// TIA Portal project "new" (V15.1)

(* hardware
DEVICE "S71500/ET200MP station_1"  S7-1500 station
   slot 0: "导轨_0"  Rack  6ES7 590-1***0-0AA0
   slot 1: "jvzihengtian"  CPU 1512C-1 PN  6ES7 512-1CK01-0AB0  V2.5
      slot 3: "CPU 显示_1"  6ES7591-1AA00-0AA0
DEVICE "DESKTOP-H96SFRB"  SIMATIC PC station
   slot 0: "SIMATIC PC station"  Rail  SIMATIC PC-Station  V1.0
      slot 125: "Stationmanager"  Station_Manager  V6.0.4
   slot 1: "IE general_1"  IE General  IE_CP  V8.2.0
   slot 2: "HMI_RT_1"  WinCC RT Advanced  6AV2 104-0xxxx-xxxx  15.1.0.0
      slot 33792: "主机接口"  Host interface
*)

// ===== PLC "jvzihengtian"  CPU 1512C-1 PN =====

DATA_BLOCK "输入变量"   // DB1
{ S7_Optimized_Access := 'FALSE' }
VERSION : 0.1
   VAR
      "1层上行呼梯按钮" : Bool;
      "2层上行呼梯按钮" : Bool;
      "3层上行呼梯按钮" : Bool;
      "4层上行呼梯按钮" : Bool;
      "5层上行呼梯按钮" : Bool;
      "2层下行呼梯按钮" : Bool;
      "3层下行呼梯按钮" : Bool;
      "4层下行呼梯按钮" : Bool;
      "5层下行呼梯按钮" : Bool;
      "6层下行呼梯按钮" : Bool;
      "1号梯轿内选层按钮1" : Bool;
      "1号梯轿内选层按钮2" : Bool;
      "1号梯轿内选层按钮3" : Bool;
      "1号梯轿内选层按钮4" : Bool;
      "1号梯轿内选层按钮5" : Bool;
      "1号梯轿内选层按钮6" : Bool;
      "1号梯轿内开门按钮" : Bool;
      "1号梯轿内关门按钮" : Bool;
      "1号梯光幕信号" : Bool;
      "1号梯检修信号" : Bool;
      "1号梯轿厢门锁信号" : Bool;
      "1号梯1楼层门锁信号" : Bool;
      "1号梯2楼层门锁信号" : Bool;
      "1号梯3楼层门锁信号" : Bool;
      "1号梯4楼层门锁信号" : Bool;
      "1号梯5楼层门锁信号" : Bool;
      "1号梯6楼层门锁信号" : Bool;
      "1号梯开门到位" : Bool;
      "1号梯关门到位" : Bool;
      "1号梯上平层信号" : Bool;
      "1号梯下平层信号" : Bool;
      "1号梯上端站第1限位" : Bool;
      "1号梯上端站第2限位" : Bool;
      "1号梯下端站第1限位" : Bool;
      "1号梯下端站第2限位" : Bool;
      自动运行信号 : Bool;
      "1号梯当前载重量" : Word;
   END_VAR
BEGIN
END_DATA_BLOCK

DATA_BLOCK "输出变量"   // DB2
{ S7_Optimized_Access := 'FALSE' }
VERSION : 0.1
   VAR
      "1层上行呼梯按钮指示灯" : Bool;
      "2层上行呼梯按钮指示灯" : Bool;
      "3层上行呼梯按钮指示灯" : Bool;
      "4层上行呼梯按钮指示灯" : Bool;
      "5层上行呼梯按钮指示灯" : Bool;
      "2层下行呼梯按钮指示灯" : Bool;
      "3层下行呼梯按钮指示灯" : Bool;
      "4层下行呼梯按钮指示灯" : Bool;
      "5层下行呼梯按钮指示灯" : Bool;
      "6层下行呼梯按钮指示灯" : Bool;
      "1号梯1层按钮指示灯" : Bool;
      "1号梯2层按钮指示灯" : Bool;
      "1号梯3层按钮指示灯" : Bool;
      "1号梯4层按钮指示灯" : Bool;
      "1号梯5层按钮指示灯" : Bool;
      "1号梯6层按钮指示灯" : Bool;
      "1号梯LEDa" : Bool;
      "1号梯LEDb" : Bool;
      "1号梯LEDc" : Bool;
      "1号梯LEDd" : Bool;
      "1号梯LEDe" : Bool;
      "1号梯LEDf" : Bool;
      "1号梯LEDg" : Bool;
      "1号梯上行指示" : Bool;
      "1号梯下行指示" : Bool;
      "1号梯故障指示" : Bool;
      "1号梯照明指示" : Bool;
      "1号梯风扇指示" : Bool;
      "1号梯满载指示" : Bool;
      "1号梯电机启动信号" : Bool := false;
      "1号梯上行接触器" : Bool;
      "1号梯下行接触器" : Bool;
      "1号梯高速接触器" : Bool;
      "1号梯低速接触器" : Bool;
      "1号梯开门继电器" : Bool;
      "1号梯关门继电器" : Bool;
      "1号梯1级减速制动" : Bool;
      "1号梯2级减速制动" : Bool;
      "1号梯3级减速制动" : Bool;
      准备就绪信号 : Bool := false;
   END_VAR
BEGIN
END_DATA_BLOCK

DATA_BLOCK "一梯辅助变量"   // DB29
{ S7_Optimized_Access := 'FALSE' }
VERSION : 0.1
   VAR
      "1层上呼tag" : Bool;
      "1层上呼开门tag" : Bool;
      "1梯关门标志" : Bool;
      "2层上呼tag" : Bool;
      "2层上呼开门tag" : Bool;
      "2层下呼tag" : Bool;
      "2层下呼开门tag" : Bool;
      "3层上呼tag" : Bool;
      "3层上呼开门tag" : Bool;
      "3层下呼tag" : Bool;
      "3层下呼开门tag" : Bool;
      "4层上呼tag" : Bool;
      "4层上呼开门tag" : Bool;
      "4层下呼tag" : Bool;
      "4层下呼开门tag" : Bool;
      "5层上呼tag" : Bool;
      "5层上呼开门tag" : Bool;
      "5层下呼tag" : Bool;
      "5层下呼开门tag" : Bool;
      "6层下呼tag" : Bool;
      "6层下呼开门tag" : Bool;
      T总延时 : Bool;
      一号梯内选1 : Bool;
      一号梯内选2 : Bool;
      一号梯内选3 : Bool;
      一号梯内选4 : Bool;
      一号梯内选5 : Bool;
      一号梯内选6 : Bool;
      一号梯初始化 : Bool;
      一号梯楼层数 : Int := 1;
      一号梯自动运行脉冲检测 : Bool;
      一层上呼标志 : Bool;
      三层上呼标志 : Bool;
      三层下呼标志 : Bool;
      "上行1，下行0，默认下" : Bool := false;
      上行标志 : Bool;
      下行标志 : Bool;
      二层上呼标志 : Bool;
      二层下呼标志 : Bool;
      五层上呼标志 : Bool;
      五层下呼标志 : Bool;
      停在1层 : Bool;
      停在2层 : Bool;
      停在3层 : Bool;
      停在4层 : Bool;
      停在5层 : Bool;
      停在6层 : Bool;
      停层信号 : Bool;
      停层关门辅助 : Bool;
      停层开门 : Bool;
      停层时上下呼开门 : Bool;
      光幕信号标志 : Bool;
      六层下呼标志 : Bool;
      关门异常重新开门 : Bool;
      关门按钮标志 : Bool;
      内选1tag : Bool;
      内选2tag : Bool;
      内选3tag : Bool;
      内选4tag : Bool;
      内选5tag : Bool;
      内选6tag : Bool;
      内选停层信号 : Bool;
      初始化上行控制 : Bool;
      初始化下行控制 : Bool;
      初始化变量1 : Bool;
      初始化变量2 : Bool;
      初始化已停层 : Bool;
      初始化平层tag : Bool;
      初始化楼层数检测 : Bool;
      到1限 : Bool;
      四层上呼标志 : Bool;
      四层下呼标志 : Bool;
      外呼停层信号 : Bool;
      延时关门辅助 : Bool;
      延时自动关门 : Bool;
      开门完成标志 : Bool;
      开门异常重新关门 : Bool;
      开门按钮标志 : Bool;
      开门标志 : Bool;
      有人出不关门 : Bool;
      楼层计数平层tag1 : Bool;
      楼层计数平层tag2 : Bool;
      超载异常强制关门 : Bool;
      超重信号 : Bool;
      超重信号tag : Bool;
      超重信号标志 : Bool;
      超重次数 : Int;
      超重次数初值 : Int;
      超重次数变化值 : Int;
      信号状态连接1 : Bool;
      载重量初值 : Word := 16#0000;
      载重变化次数计数 : Int := 0;
      载重变化一次 : Bool;
      载重变化一次tag : Bool;
      "1梯初始化到几层" : Int;
      上行1 : Bool;
      下行1 : Bool;
      上行1关 : Bool;
      下行1关 : Bool;
      上行状态检查 : Bool;
      下行状态检查 : Bool;
      上行接触器tag : Bool;
      下行接触器tag : Bool;
      上行接触器1到0 : Bool;
      下行接触器1到0 : Bool;
      开门按钮tag : Bool;
      关门按钮tag : Bool;
      光幕tag : Bool;
      "1层保护1" : Bool;
      "1层保护2" : Bool;
      "6层保护1" : Bool;
      "6层保护2" : Bool;
      内选1预消除 : Bool;
      载重量最大允许值 : Int := 13129;
      门锁状态 : Bool;
      载重变化次数max : Int := 16;
      外呼响应载重量限值 : Int := 12438;
   END_VAR
BEGIN
END_DATA_BLOCK

// folder: System blocks/Program resources

DATA_BLOCK "三级减速制动T总"   // DB3
{ S7_Optimized_Access := 'TRUE' }
AUTHOR : Simatic
FAMILY : IEC
NAME : IEC_TMR
VERSION : 1.0
// stored: InstanceOfName IEC_TIMER
"IEC_TIMER"
BEGIN
END_DATA_BLOCK

DATA_BLOCK "一级减速制动T1"   // DB4
{ S7_Optimized_Access := 'TRUE' }
AUTHOR : Simatic
FAMILY : IEC
NAME : IEC_TMR
VERSION : 1.0
// stored: InstanceOfName IEC_TIMER
"IEC_TIMER"
BEGIN
END_DATA_BLOCK

DATA_BLOCK "二级减速制动T2"   // DB5
{ S7_Optimized_Access := 'TRUE' }
AUTHOR : Simatic
FAMILY : IEC
NAME : IEC_TMR
VERSION : 1.0
// stored: InstanceOfName IEC_TIMER
"IEC_TIMER"
BEGIN
END_DATA_BLOCK

DATA_BLOCK "上下行复位脉冲"   // DB6
{ S7_Optimized_Access := 'TRUE' }
AUTHOR : Simatic
FAMILY : IEC
NAME : IEC_TMR
VERSION : 1.0
// stored: InstanceOfName IEC_TIMER
"IEC_TIMER"
BEGIN
END_DATA_BLOCK

DATA_BLOCK "初始化平层延时"   // DB7
{ S7_Optimized_Access := 'TRUE' }
AUTHOR : Simatic
FAMILY : IEC
NAME : IEC_TMR
VERSION : 1.0
// stored: InstanceOfName IEC_TIMER
"IEC_TIMER"
BEGIN
END_DATA_BLOCK

DATA_BLOCK "三级减速制动T3"   // DB8
{ S7_Optimized_Access := 'TRUE' }
AUTHOR : Simatic
FAMILY : IEC
NAME : IEC_TMR
VERSION : 1.0
// stored: InstanceOfName IEC_TIMER
"IEC_TIMER"
BEGIN
END_DATA_BLOCK

DATA_BLOCK "关断延时1"   // DB9
{ S7_Optimized_Access := 'TRUE' }
AUTHOR : Simatic
FAMILY : IEC
NAME : IEC_TMR
VERSION : 1.0
// stored: InstanceOfName IEC_TIMER
"IEC_TIMER"
BEGIN
END_DATA_BLOCK

DATA_BLOCK "停层完成延时辅助"   // DB11
{ S7_Optimized_Access := 'TRUE' }
AUTHOR : Simatic
FAMILY : IEC
NAME : IEC_TMR
VERSION : 1.0
// stored: InstanceOfName IEC_TIMER
"IEC_TIMER"
BEGIN
END_DATA_BLOCK

DATA_BLOCK "门锁好复位延时"   // DB12
{ S7_Optimized_Access := 'TRUE' }
AUTHOR : Simatic
FAMILY : IEC
NAME : IEC_TMR
VERSION : 1.0
// stored: InstanceOfName IEC_TIMER
"IEC_TIMER"
BEGIN
END_DATA_BLOCK

DATA_BLOCK "开到位延时"   // DB13
{ S7_Optimized_Access := 'TRUE' }
AUTHOR : Simatic
FAMILY : IEC
NAME : IEC_TMR
VERSION : 1.0
// stored: InstanceOfName IEC_TIMER
"IEC_TIMER"
BEGIN
END_DATA_BLOCK

DATA_BLOCK "关断延时2"   // DB14
{ S7_Optimized_Access := 'TRUE' }
AUTHOR : Simatic
FAMILY : IEC
NAME : IEC_TMR
VERSION : 1.0
// stored: InstanceOfName IEC_TIMER
"IEC_TIMER"
BEGIN
END_DATA_BLOCK

DATA_BLOCK "关断延时3"   // DB15
{ S7_Optimized_Access := 'TRUE' }
AUTHOR : Simatic
FAMILY : IEC
NAME : IEC_TMR
VERSION : 1.0
// stored: InstanceOfName IEC_TIMER
"IEC_TIMER"
BEGIN
END_DATA_BLOCK

DATA_BLOCK "关断延时4"   // DB16
{ S7_Optimized_Access := 'TRUE' }
AUTHOR : Simatic
FAMILY : IEC
NAME : IEC_TMR
VERSION : 1.0
// stored: InstanceOfName IEC_TIMER
"IEC_TIMER"
BEGIN
END_DATA_BLOCK

DATA_BLOCK "关断延时5"   // DB17
{ S7_Optimized_Access := 'TRUE' }
AUTHOR : Simatic
FAMILY : IEC
NAME : IEC_TMR
VERSION : 1.0
// stored: InstanceOfName IEC_TIMER
"IEC_TIMER"
BEGIN
END_DATA_BLOCK

DATA_BLOCK "关断延时6"   // DB18
{ S7_Optimized_Access := 'TRUE' }
AUTHOR : Simatic
FAMILY : IEC
NAME : IEC_TMR
VERSION : 1.0
// stored: InstanceOfName IEC_TIMER
"IEC_TIMER"
BEGIN
END_DATA_BLOCK

DATA_BLOCK "关断延时7"   // DB19
{ S7_Optimized_Access := 'TRUE' }
AUTHOR : Simatic
FAMILY : IEC
NAME : IEC_TMR
VERSION : 1.0
// stored: InstanceOfName IEC_TIMER
"IEC_TIMER"
BEGIN
END_DATA_BLOCK

DATA_BLOCK "待载休眠计时"   // DB20
{ S7_Optimized_Access := 'TRUE' }
AUTHOR : Simatic
FAMILY : IEC
NAME : IEC_TMR
VERSION : 1.0
// stored: InstanceOfName IEC_TIMER
"IEC_TIMER"
BEGIN
END_DATA_BLOCK

DATA_BLOCK "关门时间"   // DB21
{ S7_Optimized_Access := 'TRUE' }
AUTHOR : Simatic
FAMILY : IEC
NAME : IEC_TMR
VERSION : 1.0
// stored: InstanceOfName IEC_TIMER
"IEC_TIMER"
BEGIN
END_DATA_BLOCK

DATA_BLOCK "关断延时8"   // DB22
{ S7_Optimized_Access := 'TRUE' }
AUTHOR : Simatic
FAMILY : IEC
NAME : IEC_TMR
VERSION : 1.0
// stored: InstanceOfName IEC_TIMER
"IEC_TIMER"
BEGIN
END_DATA_BLOCK

DATA_BLOCK "超重延时判断"   // DB23
{ S7_Optimized_Access := 'TRUE' }
AUTHOR : Simatic
FAMILY : IEC
NAME : IEC_TMR
VERSION : 1.0
// stored: InstanceOfName IEC_TIMER
"IEC_TIMER"
BEGIN
END_DATA_BLOCK

DATA_BLOCK "超载异常脉冲"   // DB24
{ S7_Optimized_Access := 'TRUE' }
AUTHOR : Simatic
FAMILY : IEC
NAME : IEC_TMR
VERSION : 1.0
// stored: InstanceOfName IEC_TIMER
"IEC_TIMER"
BEGIN
END_DATA_BLOCK

DATA_BLOCK "关断延时9"   // DB25
{ S7_Optimized_Access := 'TRUE' }
AUTHOR : Simatic
FAMILY : IEC
NAME : IEC_TMR
VERSION : 1.0
// stored: InstanceOfName IEC_TIMER
"IEC_TIMER"
BEGIN
END_DATA_BLOCK

DATA_BLOCK "低速启动延时"   // DB26
{ S7_Optimized_Access := 'TRUE' }
AUTHOR : Simatic
FAMILY : IEC
NAME : IEC_TMR
VERSION : 1.0
// stored: InstanceOfName IEC_TIMER
"IEC_TIMER"
BEGIN
END_DATA_BLOCK

DATA_BLOCK "关断延时10"   // DB27
{ S7_Optimized_Access := 'TRUE' }
AUTHOR : Simatic
FAMILY : IEC
NAME : IEC_TMR
VERSION : 1.0
// stored: InstanceOfName IEC_TIMER
"IEC_TIMER"
BEGIN
END_DATA_BLOCK

DATA_BLOCK "开门时间"   // DB28
{ S7_Optimized_Access := 'TRUE' }
AUTHOR : Simatic
FAMILY : IEC
NAME : IEC_TMR
VERSION : 1.0
// stored: InstanceOfName IEC_TIMER
"IEC_TIMER"
BEGIN
END_DATA_BLOCK

DATA_BLOCK "载重量比较"   // DB30
{ S7_Optimized_Access := 'TRUE' }
AUTHOR : Simatic
FAMILY : IEC
NAME : IEC_TMR
VERSION : 1.0
// stored: InstanceOfName IEC_TIMER
"IEC_TIMER"
BEGIN
END_DATA_BLOCK

DATA_BLOCK "采样、比较时间间隔"   // DB31
{ S7_Optimized_Access := 'TRUE' }
AUTHOR : Simatic
FAMILY : IEC
NAME : IEC_TMR
VERSION : 1.0
// stored: InstanceOfName IEC_TIMER
"IEC_TIMER"
BEGIN
END_DATA_BLOCK

DATA_BLOCK "载重量采样"   // DB32
{ S7_Optimized_Access := 'TRUE' }
AUTHOR : Simatic
FAMILY : IEC
NAME : IEC_TMR
VERSION : 1.0
// stored: InstanceOfName IEC_TIMER
"IEC_TIMER"
BEGIN
END_DATA_BLOCK

DATA_BLOCK "关断延时11"   // DB33
{ S7_Optimized_Access := 'TRUE' }
AUTHOR : Simatic
FAMILY : IEC
NAME : IEC_TMR
VERSION : 1.0
// stored: InstanceOfName IEC_TIMER
"IEC_TIMER"
BEGIN
END_DATA_BLOCK

DATA_BLOCK "IEC_Timer_0_DB_4"   // DB34
{ S7_Optimized_Access := 'TRUE' }
AUTHOR : Simatic
FAMILY : IEC
NAME : IEC_TMR
VERSION : 1.0
// stored: InstanceOfName IEC_TIMER
"IEC_TIMER"
BEGIN
END_DATA_BLOCK

DATA_BLOCK "关断延时12"   // DB35
{ S7_Optimized_Access := 'TRUE' }
AUTHOR : Simatic
FAMILY : IEC
NAME : IEC_TMR
VERSION : 1.0
// stored: InstanceOfName IEC_TIMER
"IEC_TIMER"
BEGIN
END_DATA_BLOCK

DATA_BLOCK "关断延时13"   // DB36
{ S7_Optimized_Access := 'TRUE' }
AUTHOR : Simatic
FAMILY : IEC
NAME : IEC_TMR
VERSION : 1.0
// stored: InstanceOfName IEC_TIMER
"IEC_TIMER"
BEGIN
END_DATA_BLOCK

DATA_BLOCK "关断延时14"   // DB37
{ S7_Optimized_Access := 'TRUE' }
AUTHOR : Simatic
FAMILY : IEC
NAME : IEC_TMR
VERSION : 1.0
// stored: InstanceOfName IEC_TIMER
"IEC_TIMER"
BEGIN
END_DATA_BLOCK

DATA_BLOCK "关断延时15"   // DB38
{ S7_Optimized_Access := 'TRUE' }
AUTHOR : Simatic
FAMILY : IEC
NAME : IEC_TMR
VERSION : 1.0
// stored: InstanceOfName IEC_TIMER
"IEC_TIMER"
BEGIN
END_DATA_BLOCK

DATA_BLOCK "关断延时16"   // DB39
{ S7_Optimized_Access := 'TRUE' }
AUTHOR : Simatic
FAMILY : IEC
NAME : IEC_TMR
VERSION : 1.0
// stored: InstanceOfName IEC_TIMER
"IEC_TIMER"
BEGIN
END_DATA_BLOCK

DATA_BLOCK "计数"   // DB40
{ S7_Optimized_Access := 'TRUE' }
AUTHOR : Simatic
FAMILY : IEC
NAME : CNTR
VERSION : 1.0
// stored: InstanceOfName IEC_COUNTER
"IEC_COUNTER"
BEGIN
END_DATA_BLOCK

DATA_BLOCK "内选错误消除限时"   // DB50
{ S7_Optimized_Access := 'TRUE' }
AUTHOR : Simatic
FAMILY : IEC
NAME : IEC_TMR
VERSION : 1.0
// stored: InstanceOfName IEC_TIMER
"IEC_TIMER"
BEGIN
END_DATA_BLOCK

DATA_BLOCK "消除标志复位"   // DB51
{ S7_Optimized_Access := 'TRUE' }
AUTHOR : Simatic
FAMILY : IEC
NAME : IEC_TMR
VERSION : 1.0
// stored: InstanceOfName IEC_TIMER
"IEC_TIMER"
BEGIN
END_DATA_BLOCK

DATA_BLOCK "消除延时"   // DB52
{ S7_Optimized_Access := 'TRUE' }
AUTHOR : Simatic
FAMILY : IEC
NAME : IEC_TMR
VERSION : 1.0
// stored: InstanceOfName IEC_TIMER
"IEC_TIMER"
BEGIN
END_DATA_BLOCK

// folder: (top level)

FUNCTION "初始化下行" : Void   // FC1, LAD
{ S7_Optimized_Access := 'TRUE' }
VERSION : 0.1
   VAR_TEMP   // added for the SCL form of the ladder/FBD networks
      _w1 : Bool;
   END_VAR
BEGIN

REGION Network 1: 下行初始化
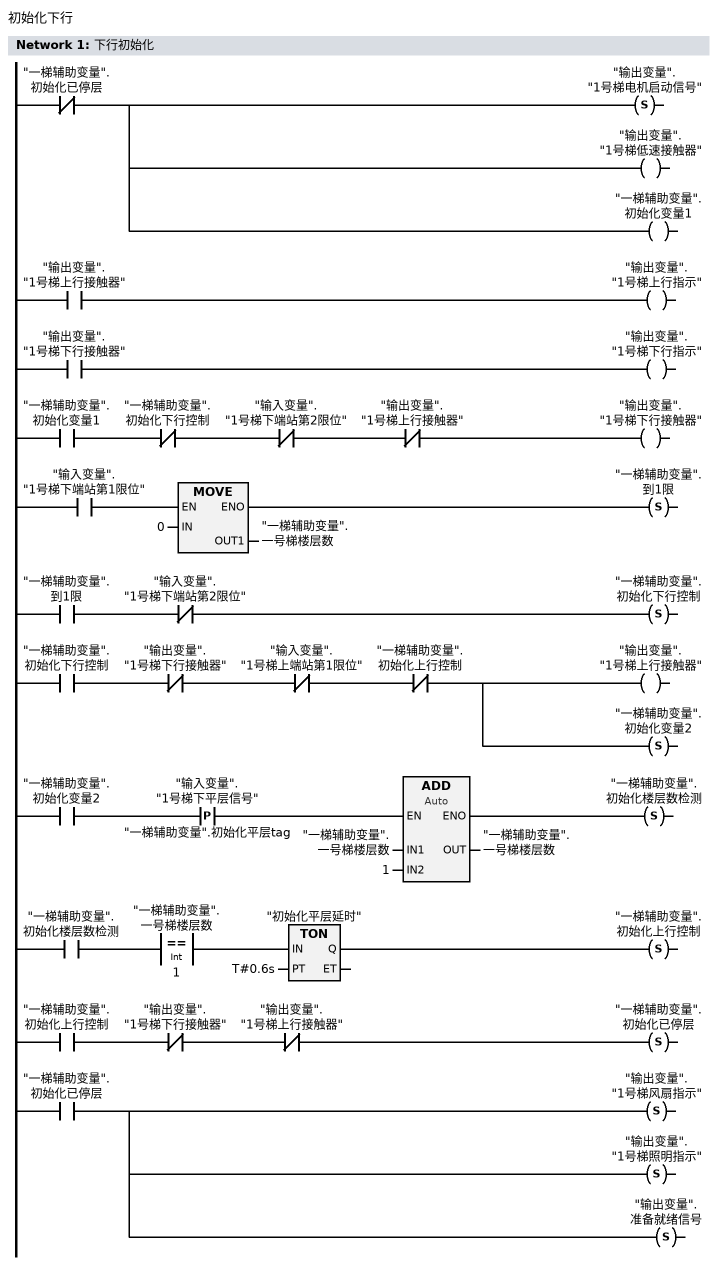
   IF NOT "一梯辅助变量".初始化已停层 THEN "输出变量"."1号梯电机启动信号" := TRUE; END_IF;
   "输出变量"."1号梯低速接触器" := NOT "一梯辅助变量".初始化已停层;
   "一梯辅助变量".初始化变量1 := NOT "一梯辅助变量".初始化已停层;
   "输出变量"."1号梯上行指示" := "输出变量"."1号梯上行接触器";
   "输出变量"."1号梯下行指示" := "输出变量"."1号梯下行接触器";
   "输出变量"."1号梯下行接触器" := "一梯辅助变量".初始化变量1 AND NOT "一梯辅助变量".初始化下行控制 AND NOT "输入变量"."1号梯下端站第2限位" AND NOT "输出变量"."1号梯上行接触器";
   IF "输入变量"."1号梯下端站第1限位" THEN
       "一梯辅助变量".一号梯楼层数 := 0;
       "一梯辅助变量".到1限 := TRUE;
   END_IF;
   IF "一梯辅助变量".到1限 AND NOT "输入变量"."1号梯下端站第2限位" THEN "一梯辅助变量".初始化下行控制 := TRUE; END_IF;
   "输出变量"."1号梯上行接触器" := "一梯辅助变量".初始化下行控制 AND NOT "输出变量"."1号梯下行接触器" AND NOT "输入变量"."1号梯上端站第1限位" AND NOT "一梯辅助变量".初始化上行控制;
   IF "输出变量"."1号梯上行接触器" THEN "一梯辅助变量".初始化变量2 := TRUE; END_IF;
   #_w1 := "一梯辅助变量".初始化变量2 AND "输入变量"."1号梯下平层信号" AND NOT "一梯辅助变量".初始化平层tag;   // rising edge of "输入变量"."1号梯下平层信号"
   "一梯辅助变量".初始化平层tag := "输入变量"."1号梯下平层信号";
   IF #_w1 THEN
       "一梯辅助变量".一号梯楼层数 := "一梯辅助变量".一号梯楼层数 + 1;
       "一梯辅助变量".初始化楼层数检测 := TRUE;
   END_IF;
   "初始化平层延时".TON(IN := "一梯辅助变量".初始化楼层数检测 AND ("一梯辅助变量".一号梯楼层数 = 1), PT := T#0.6s);
   IF "初始化平层延时".Q THEN "一梯辅助变量".初始化上行控制 := TRUE; END_IF;
   IF "一梯辅助变量".初始化上行控制 AND NOT "输出变量"."1号梯下行接触器" AND NOT "输出变量"."1号梯上行接触器" THEN
       "一梯辅助变量".初始化已停层 := TRUE;
   END_IF;
   IF "一梯辅助变量".初始化已停层 THEN
       "输出变量"."1号梯风扇指示" := TRUE;
       "输出变量"."1号梯照明指示" := TRUE;
       "输出变量".准备就绪信号 := TRUE;
   END_IF;
END_REGION
END_FUNCTION

FUNCTION "呼梯信号" : Void   // FC2, LAD
{ S7_Optimized_Access := 'TRUE' }
VERSION : 0.1
   VAR_TEMP   // added for the SCL form of the ladder/FBD networks
      _w1 : Bool;
      _w2 : Bool;
      _w3 : Bool;
      _w4 : Bool;
      _w5 : Bool;
      _w6 : Bool;
      _w7 : Bool;
      _w8 : Bool;
      _w9 : Bool;
      _w10 : Bool;
      _w11 : Bool;
      _w12 : Bool;
   END_VAR
BEGIN

REGION Network 1: 外呼灯
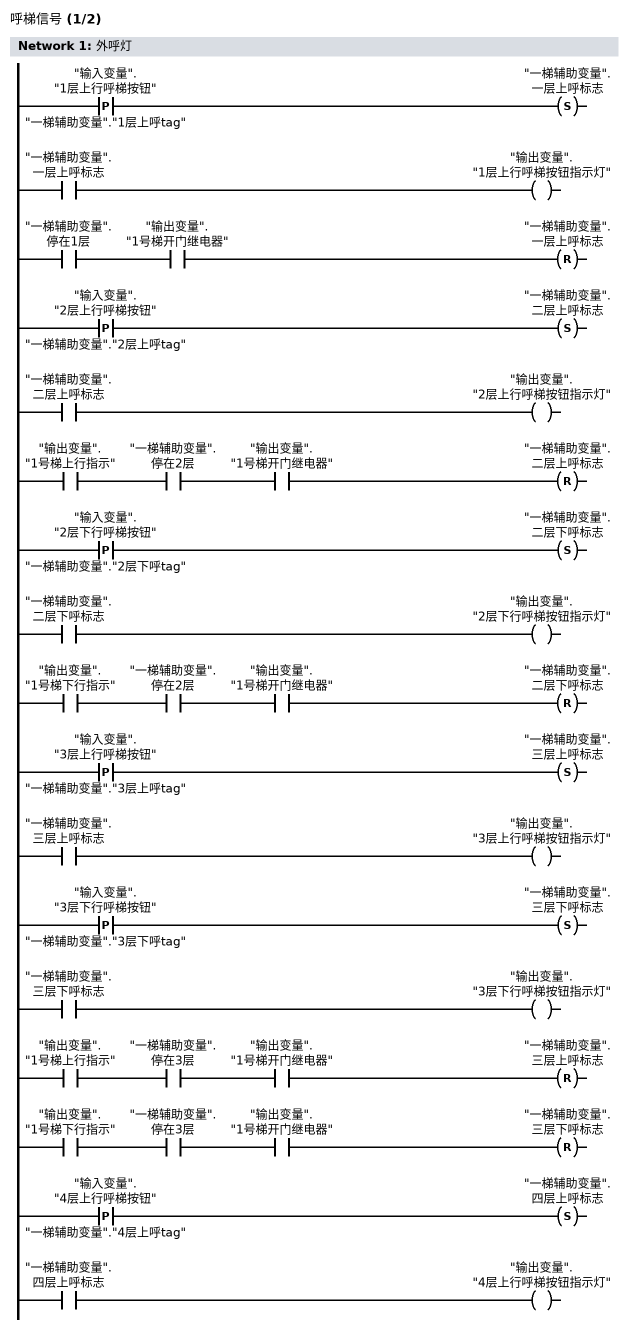
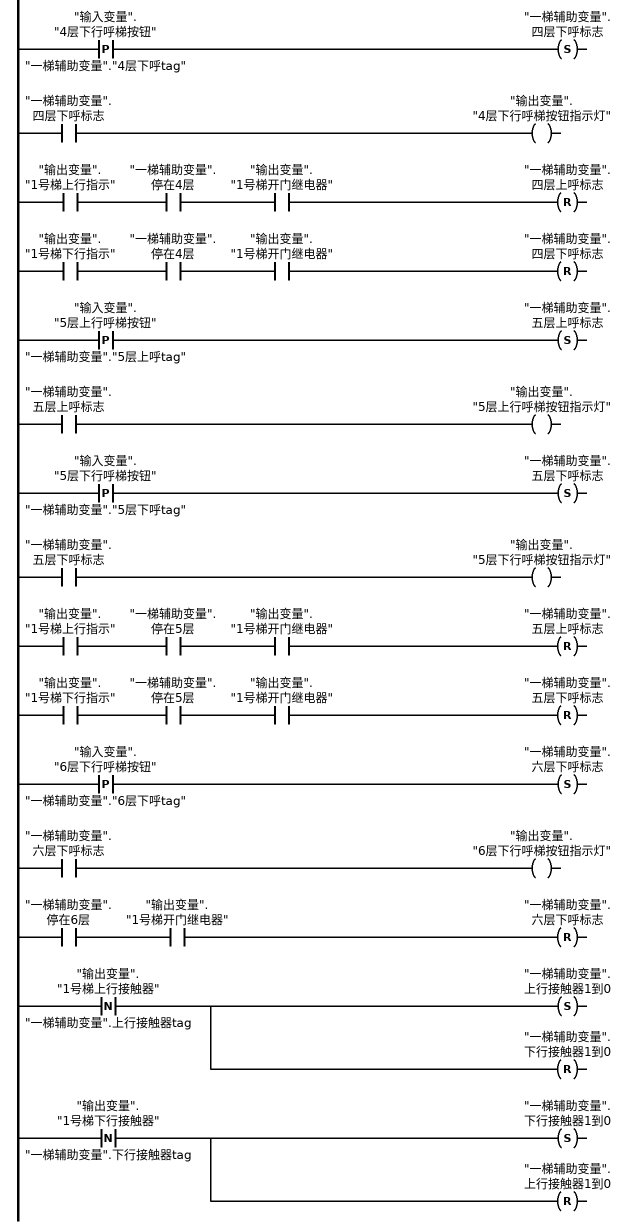
   RUNG wire#powerrail
      P_Contact(operand := "输入变量"."1层上行呼梯按钮", bit := "一梯辅助变量"."1层上呼tag")
      S_Coil( "一梯辅助变量".一层上呼标志 )
   END_RUNG
   RUNG wire#powerrail
      Contact( "一梯辅助变量".一层上呼标志 )
      Coil( "输出变量"."1层上行呼梯按钮指示灯" )
   END_RUNG
   RUNG wire#powerrail
      Contact( "一梯辅助变量".停在1层 )
      Contact( "输出变量"."1号梯开门继电器" )
      R_Coil( "一梯辅助变量".一层上呼标志 )
   END_RUNG
   RUNG wire#powerrail
      P_Contact(operand := "输入变量"."2层上行呼梯按钮", bit := "一梯辅助变量"."2层上呼tag")
      S_Coil( "一梯辅助变量".二层上呼标志 )
   END_RUNG
   RUNG wire#powerrail
      Contact( "一梯辅助变量".二层上呼标志 )
      Coil( "输出变量"."2层上行呼梯按钮指示灯" )
   END_RUNG
   RUNG wire#powerrail
      Contact( "输出变量"."1号梯上行指示" )
      Contact( "一梯辅助变量".停在2层 )
      Contact( "输出变量"."1号梯开门继电器" )
      R_Coil( "一梯辅助变量".二层上呼标志 )
   END_RUNG
   RUNG wire#powerrail
      P_Contact(operand := "输入变量"."2层下行呼梯按钮", bit := "一梯辅助变量"."2层下呼tag")
      S_Coil( "一梯辅助变量".二层下呼标志 )
   END_RUNG
   RUNG wire#powerrail
      Contact( "一梯辅助变量".二层下呼标志 )
      Coil( "输出变量"."2层下行呼梯按钮指示灯" )
   END_RUNG
   RUNG wire#powerrail
      Contact( "输出变量"."1号梯下行指示" )
      Contact( "一梯辅助变量".停在2层 )
      Contact( "输出变量"."1号梯开门继电器" )
      R_Coil( "一梯辅助变量".二层下呼标志 )
   END_RUNG
   RUNG wire#powerrail
      P_Contact(operand := "输入变量"."3层上行呼梯按钮", bit := "一梯辅助变量"."3层上呼tag")
      S_Coil( "一梯辅助变量".三层上呼标志 )
   END_RUNG
   RUNG wire#powerrail
      Contact( "一梯辅助变量".三层上呼标志 )
      Coil( "输出变量"."3层上行呼梯按钮指示灯" )
   END_RUNG
   RUNG wire#powerrail
      P_Contact(operand := "输入变量"."3层下行呼梯按钮", bit := "一梯辅助变量"."3层下呼tag")
      S_Coil( "一梯辅助变量".三层下呼标志 )
   END_RUNG
   RUNG wire#powerrail
      Contact( "一梯辅助变量".三层下呼标志 )
      Coil( "输出变量"."3层下行呼梯按钮指示灯" )
   END_RUNG
   RUNG wire#powerrail
      Contact( "输出变量"."1号梯上行指示" )
      Contact( "一梯辅助变量".停在3层 )
      Contact( "输出变量"."1号梯开门继电器" )
      R_Coil( "一梯辅助变量".三层上呼标志 )
   END_RUNG
   RUNG wire#powerrail
      Contact( "输出变量"."1号梯下行指示" )
      Contact( "一梯辅助变量".停在3层 )
      Contact( "输出变量"."1号梯开门继电器" )
      R_Coil( "一梯辅助变量".三层下呼标志 )
   END_RUNG
   RUNG wire#powerrail
      P_Contact(operand := "输入变量"."4层上行呼梯按钮", bit := "一梯辅助变量"."4层上呼tag")
      S_Coil( "一梯辅助变量".四层上呼标志 )
   END_RUNG
   RUNG wire#powerrail
      Contact( "一梯辅助变量".四层上呼标志 )
      Coil( "输出变量"."4层上行呼梯按钮指示灯" )
   END_RUNG
   RUNG wire#powerrail
      P_Contact(operand := "输入变量"."4层下行呼梯按钮", bit := "一梯辅助变量"."4层下呼tag")
      S_Coil( "一梯辅助变量".四层下呼标志 )
   END_RUNG
   RUNG wire#powerrail
      Contact( "一梯辅助变量".四层下呼标志 )
      Coil( "输出变量"."4层下行呼梯按钮指示灯" )
   END_RUNG
   RUNG wire#powerrail
      Contact( "输出变量"."1号梯上行指示" )
      Contact( "一梯辅助变量".停在4层 )
      Contact( "输出变量"."1号梯开门继电器" )
      R_Coil( "一梯辅助变量".四层上呼标志 )
   END_RUNG
   RUNG wire#powerrail
      Contact( "输出变量"."1号梯下行指示" )
      Contact( "一梯辅助变量".停在4层 )
      Contact( "输出变量"."1号梯开门继电器" )
      R_Coil( "一梯辅助变量".四层下呼标志 )
   END_RUNG
   RUNG wire#powerrail
      P_Contact(operand := "输入变量"."5层上行呼梯按钮", bit := "一梯辅助变量"."5层上呼tag")
      S_Coil( "一梯辅助变量".五层上呼标志 )
   END_RUNG
   RUNG wire#powerrail
      Contact( "一梯辅助变量".五层上呼标志 )
      Coil( "输出变量"."5层上行呼梯按钮指示灯" )
   END_RUNG
   RUNG wire#powerrail
      P_Contact(operand := "输入变量"."5层下行呼梯按钮", bit := "一梯辅助变量"."5层下呼tag")
      S_Coil( "一梯辅助变量".五层下呼标志 )
   END_RUNG
   RUNG wire#powerrail
      Contact( "一梯辅助变量".五层下呼标志 )
      Coil( "输出变量"."5层下行呼梯按钮指示灯" )
   END_RUNG
   RUNG wire#powerrail
      Contact( "输出变量"."1号梯上行指示" )
      Contact( "一梯辅助变量".停在5层 )
      Contact( "输出变量"."1号梯开门继电器" )
      R_Coil( "一梯辅助变量".五层上呼标志 )
   END_RUNG
   RUNG wire#powerrail
      Contact( "输出变量"."1号梯下行指示" )
      Contact( "一梯辅助变量".停在5层 )
      Contact( "输出变量"."1号梯开门继电器" )
      R_Coil( "一梯辅助变量".五层下呼标志 )
   END_RUNG
   RUNG wire#powerrail
      P_Contact(operand := "输入变量"."6层下行呼梯按钮", bit := "一梯辅助变量"."6层下呼tag")
      S_Coil( "一梯辅助变量".六层下呼标志 )
   END_RUNG
   RUNG wire#powerrail
      Contact( "一梯辅助变量".六层下呼标志 )
      Coil( "输出变量"."6层下行呼梯按钮指示灯" )
   END_RUNG
   RUNG wire#powerrail
      Contact( "一梯辅助变量".停在6层 )
      Contact( "输出变量"."1号梯开门继电器" )
      R_Coil( "一梯辅助变量".六层下呼标志 )
   END_RUNG
   RUNG wire#powerrail
      N_Contact(operand := "输出变量"."1号梯上行接触器", bit := "一梯辅助变量".上行接触器tag)
      wire#w1
      S_Coil( "一梯辅助变量".上行接触器1到0 )
   END_RUNG
   RUNG wire#w1
      R_Coil( "一梯辅助变量".下行接触器1到0 )
   END_RUNG
   RUNG wire#powerrail
      N_Contact(operand := "输出变量"."1号梯下行接触器", bit := "一梯辅助变量".下行接触器tag)
      wire#w2
      S_Coil( "一梯辅助变量".下行接触器1到0 )
   END_RUNG
   RUNG wire#w2
      R_Coil( "一梯辅助变量".上行接触器1到0 )
   END_RUNG
   // the same network as SCL:
   #_w1 := "输入变量"."1层上行呼梯按钮" AND NOT "一梯辅助变量"."1层上呼tag";   // rising edge of "输入变量"."1层上行呼梯按钮"
   "一梯辅助变量"."1层上呼tag" := "输入变量"."1层上行呼梯按钮";
   IF #_w1 THEN "一梯辅助变量".一层上呼标志 := TRUE; END_IF;
   "输出变量"."1层上行呼梯按钮指示灯" := "一梯辅助变量".一层上呼标志;
   IF "一梯辅助变量".停在1层 AND "输出变量"."1号梯开门继电器" THEN "一梯辅助变量".一层上呼标志 := FALSE; END_IF;
   #_w2 := "输入变量"."2层上行呼梯按钮" AND NOT "一梯辅助变量"."2层上呼tag";   // rising edge of "输入变量"."2层上行呼梯按钮"
   "一梯辅助变量"."2层上呼tag" := "输入变量"."2层上行呼梯按钮";
   IF #_w2 THEN "一梯辅助变量".二层上呼标志 := TRUE; END_IF;
   "输出变量"."2层上行呼梯按钮指示灯" := "一梯辅助变量".二层上呼标志;
   IF "输出变量"."1号梯上行指示" AND "一梯辅助变量".停在2层 AND "输出变量"."1号梯开门继电器" THEN "一梯辅助变量".二层上呼标志 := FALSE; END_IF;
   #_w3 := "输入变量"."2层下行呼梯按钮" AND NOT "一梯辅助变量"."2层下呼tag";   // rising edge of "输入变量"."2层下行呼梯按钮"
   "一梯辅助变量"."2层下呼tag" := "输入变量"."2层下行呼梯按钮";
   IF #_w3 THEN "一梯辅助变量".二层下呼标志 := TRUE; END_IF;
   "输出变量"."2层下行呼梯按钮指示灯" := "一梯辅助变量".二层下呼标志;
   IF "输出变量"."1号梯下行指示" AND "一梯辅助变量".停在2层 AND "输出变量"."1号梯开门继电器" THEN "一梯辅助变量".二层下呼标志 := FALSE; END_IF;
   #_w4 := "输入变量"."3层上行呼梯按钮" AND NOT "一梯辅助变量"."3层上呼tag";   // rising edge of "输入变量"."3层上行呼梯按钮"
   "一梯辅助变量"."3层上呼tag" := "输入变量"."3层上行呼梯按钮";
   IF #_w4 THEN "一梯辅助变量".三层上呼标志 := TRUE; END_IF;
   "输出变量"."3层上行呼梯按钮指示灯" := "一梯辅助变量".三层上呼标志;
   #_w5 := "输入变量"."3层下行呼梯按钮" AND NOT "一梯辅助变量"."3层下呼tag";   // rising edge of "输入变量"."3层下行呼梯按钮"
   "一梯辅助变量"."3层下呼tag" := "输入变量"."3层下行呼梯按钮";
   IF #_w5 THEN "一梯辅助变量".三层下呼标志 := TRUE; END_IF;
   "输出变量"."3层下行呼梯按钮指示灯" := "一梯辅助变量".三层下呼标志;
   IF "输出变量"."1号梯上行指示" AND "一梯辅助变量".停在3层 AND "输出变量"."1号梯开门继电器" THEN "一梯辅助变量".三层上呼标志 := FALSE; END_IF;
   IF "输出变量"."1号梯下行指示" AND "一梯辅助变量".停在3层 AND "输出变量"."1号梯开门继电器" THEN "一梯辅助变量".三层下呼标志 := FALSE; END_IF;
   #_w6 := "输入变量"."4层上行呼梯按钮" AND NOT "一梯辅助变量"."4层上呼tag";   // rising edge of "输入变量"."4层上行呼梯按钮"
   "一梯辅助变量"."4层上呼tag" := "输入变量"."4层上行呼梯按钮";
   IF #_w6 THEN "一梯辅助变量".四层上呼标志 := TRUE; END_IF;
   "输出变量"."4层上行呼梯按钮指示灯" := "一梯辅助变量".四层上呼标志;
   #_w7 := "输入变量"."4层下行呼梯按钮" AND NOT "一梯辅助变量"."4层下呼tag";   // rising edge of "输入变量"."4层下行呼梯按钮"
   "一梯辅助变量"."4层下呼tag" := "输入变量"."4层下行呼梯按钮";
   IF #_w7 THEN "一梯辅助变量".四层下呼标志 := TRUE; END_IF;
   "输出变量"."4层下行呼梯按钮指示灯" := "一梯辅助变量".四层下呼标志;
   IF "输出变量"."1号梯上行指示" AND "一梯辅助变量".停在4层 AND "输出变量"."1号梯开门继电器" THEN "一梯辅助变量".四层上呼标志 := FALSE; END_IF;
   IF "输出变量"."1号梯下行指示" AND "一梯辅助变量".停在4层 AND "输出变量"."1号梯开门继电器" THEN "一梯辅助变量".四层下呼标志 := FALSE; END_IF;
   #_w8 := "输入变量"."5层上行呼梯按钮" AND NOT "一梯辅助变量"."5层上呼tag";   // rising edge of "输入变量"."5层上行呼梯按钮"
   "一梯辅助变量"."5层上呼tag" := "输入变量"."5层上行呼梯按钮";
   IF #_w8 THEN "一梯辅助变量".五层上呼标志 := TRUE; END_IF;
   "输出变量"."5层上行呼梯按钮指示灯" := "一梯辅助变量".五层上呼标志;
   #_w9 := "输入变量"."5层下行呼梯按钮" AND NOT "一梯辅助变量"."5层下呼tag";   // rising edge of "输入变量"."5层下行呼梯按钮"
   "一梯辅助变量"."5层下呼tag" := "输入变量"."5层下行呼梯按钮";
   IF #_w9 THEN "一梯辅助变量".五层下呼标志 := TRUE; END_IF;
   "输出变量"."5层下行呼梯按钮指示灯" := "一梯辅助变量".五层下呼标志;
   IF "输出变量"."1号梯上行指示" AND "一梯辅助变量".停在5层 AND "输出变量"."1号梯开门继电器" THEN "一梯辅助变量".五层上呼标志 := FALSE; END_IF;
   IF "输出变量"."1号梯下行指示" AND "一梯辅助变量".停在5层 AND "输出变量"."1号梯开门继电器" THEN "一梯辅助变量".五层下呼标志 := FALSE; END_IF;
   #_w10 := "输入变量"."6层下行呼梯按钮" AND NOT "一梯辅助变量"."6层下呼tag";   // rising edge of "输入变量"."6层下行呼梯按钮"
   "一梯辅助变量"."6层下呼tag" := "输入变量"."6层下行呼梯按钮";
   IF #_w10 THEN "一梯辅助变量".六层下呼标志 := TRUE; END_IF;
   "输出变量"."6层下行呼梯按钮指示灯" := "一梯辅助变量".六层下呼标志;
   IF "一梯辅助变量".停在6层 AND "输出变量"."1号梯开门继电器" THEN "一梯辅助变量".六层下呼标志 := FALSE; END_IF;
   #_w11 := NOT "输出变量"."1号梯上行接触器" AND "一梯辅助变量".上行接触器tag;   // falling edge of "输出变量"."1号梯上行接触器"
   "一梯辅助变量".上行接触器tag := "输出变量"."1号梯上行接触器";
   IF #_w11 THEN
       "一梯辅助变量".上行接触器1到0 := TRUE;
       "一梯辅助变量".下行接触器1到0 := FALSE;
   END_IF;
   #_w12 := NOT "输出变量"."1号梯下行接触器" AND "一梯辅助变量".下行接触器tag;   // falling edge of "输出变量"."1号梯下行接触器"
   "一梯辅助变量".下行接触器tag := "输出变量"."1号梯下行接触器";
   IF #_w12 THEN
       "一梯辅助变量".下行接触器1到0 := TRUE;
       "一梯辅助变量".上行接触器1到0 := FALSE;
   END_IF;
END_REGION

REGION Network 2: 内选灯
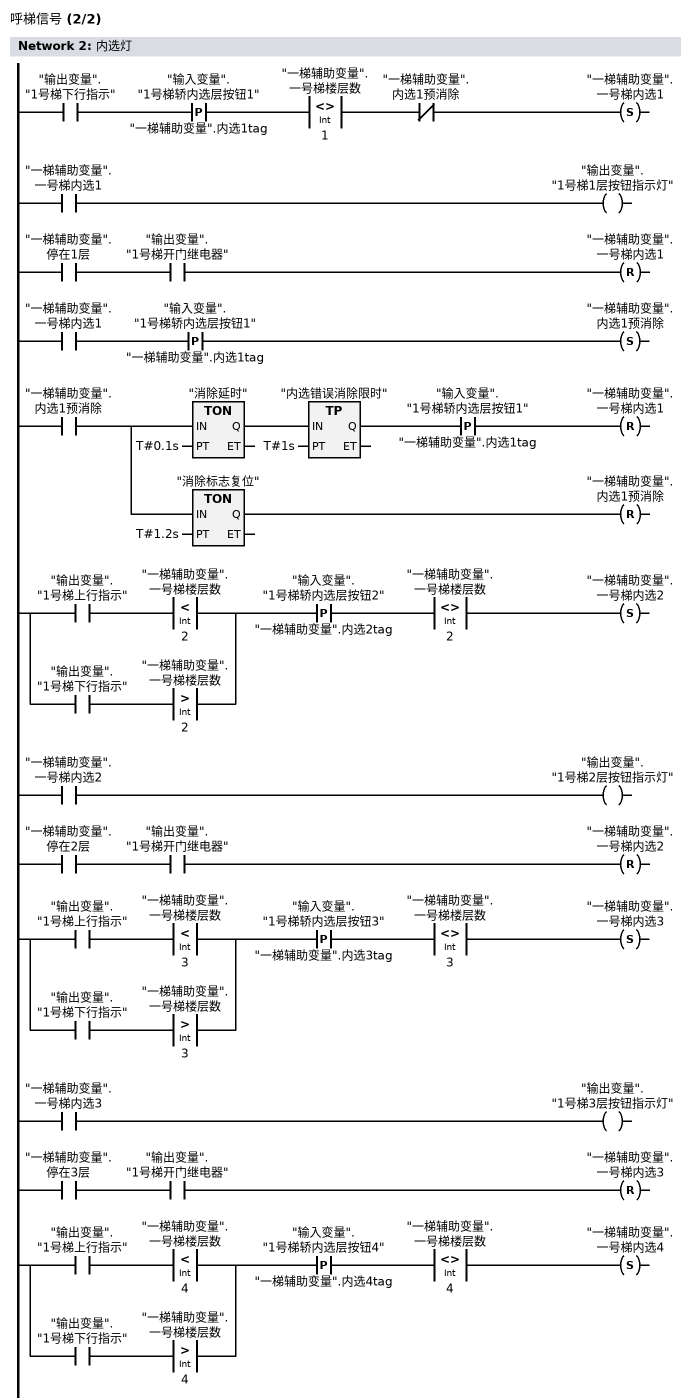
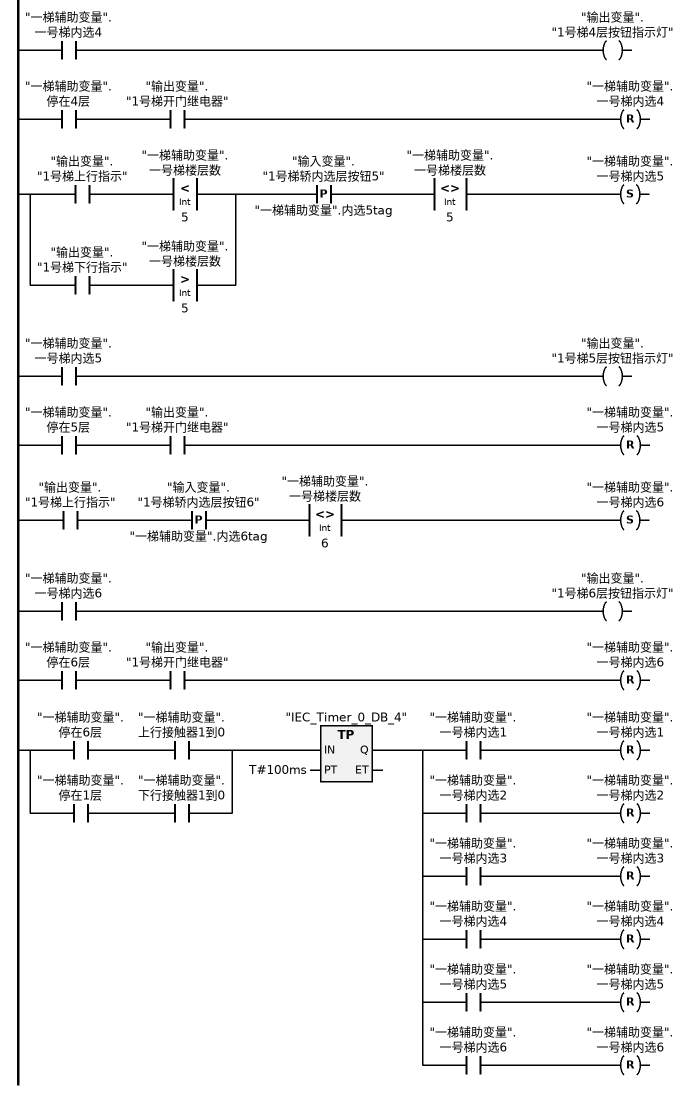
   #_w1 := "输出变量"."1号梯下行指示" AND "输入变量"."1号梯轿内选层按钮1" AND NOT "一梯辅助变量".内选1tag;   // rising edge of "输入变量"."1号梯轿内选层按钮1"
   "一梯辅助变量".内选1tag := "输入变量"."1号梯轿内选层按钮1";
   IF #_w1 AND ("一梯辅助变量".一号梯楼层数 <> 1) AND NOT "一梯辅助变量".内选1预消除 THEN "一梯辅助变量".一号梯内选1 := TRUE; END_IF;
   "输出变量"."1号梯1层按钮指示灯" := "一梯辅助变量".一号梯内选1;
   IF "一梯辅助变量".停在1层 AND "输出变量"."1号梯开门继电器" THEN "一梯辅助变量".一号梯内选1 := FALSE; END_IF;
   #_w2 := "一梯辅助变量".一号梯内选1 AND "输入变量"."1号梯轿内选层按钮1" AND NOT "一梯辅助变量".内选1tag;   // rising edge of "输入变量"."1号梯轿内选层按钮1"
   "一梯辅助变量".内选1tag := "输入变量"."1号梯轿内选层按钮1";
   IF #_w2 THEN "一梯辅助变量".内选1预消除 := TRUE; END_IF;
   "消除延时".TON(IN := "一梯辅助变量".内选1预消除, PT := T#0.1s);
   "内选错误消除限时".TP(IN := "消除延时".Q, PT := T#1s);
   #_w3 := "内选错误消除限时".Q AND "输入变量"."1号梯轿内选层按钮1" AND NOT "一梯辅助变量".内选1tag;   // rising edge of "输入变量"."1号梯轿内选层按钮1"
   "一梯辅助变量".内选1tag := "输入变量"."1号梯轿内选层按钮1";
   IF #_w3 THEN "一梯辅助变量".一号梯内选1 := FALSE; END_IF;
   "消除标志复位".TON(IN := "一梯辅助变量".内选1预消除, PT := T#1.2s);
   IF "消除标志复位".Q THEN "一梯辅助变量".内选1预消除 := FALSE; END_IF;
   #_w4 := (("输出变量"."1号梯上行指示" AND ("一梯辅助变量".一号梯楼层数 < 2)) OR ("输出变量"."1号梯下行指示" AND ("一梯辅助变量".一号梯楼层数 > 2))) AND "输入变量"."1号梯轿内选层按钮2" AND NOT "一梯辅助变量".内选2tag;   // rising edge of "输入变量"."1号梯轿内选层按钮2"
   "一梯辅助变量".内选2tag := "输入变量"."1号梯轿内选层按钮2";
   IF #_w4 AND ("一梯辅助变量".一号梯楼层数 <> 2) THEN "一梯辅助变量".一号梯内选2 := TRUE; END_IF;
   "输出变量"."1号梯2层按钮指示灯" := "一梯辅助变量".一号梯内选2;
   IF "一梯辅助变量".停在2层 AND "输出变量"."1号梯开门继电器" THEN "一梯辅助变量".一号梯内选2 := FALSE; END_IF;
   #_w5 := (("输出变量"."1号梯上行指示" AND ("一梯辅助变量".一号梯楼层数 < 3)) OR ("输出变量"."1号梯下行指示" AND ("一梯辅助变量".一号梯楼层数 > 3))) AND "输入变量"."1号梯轿内选层按钮3" AND NOT "一梯辅助变量".内选3tag;   // rising edge of "输入变量"."1号梯轿内选层按钮3"
   "一梯辅助变量".内选3tag := "输入变量"."1号梯轿内选层按钮3";
   IF #_w5 AND ("一梯辅助变量".一号梯楼层数 <> 3) THEN "一梯辅助变量".一号梯内选3 := TRUE; END_IF;
   "输出变量"."1号梯3层按钮指示灯" := "一梯辅助变量".一号梯内选3;
   IF "一梯辅助变量".停在3层 AND "输出变量"."1号梯开门继电器" THEN "一梯辅助变量".一号梯内选3 := FALSE; END_IF;
   #_w6 := (("输出变量"."1号梯上行指示" AND ("一梯辅助变量".一号梯楼层数 < 4)) OR ("输出变量"."1号梯下行指示" AND ("一梯辅助变量".一号梯楼层数 > 4))) AND "输入变量"."1号梯轿内选层按钮4" AND NOT "一梯辅助变量".内选4tag;   // rising edge of "输入变量"."1号梯轿内选层按钮4"
   "一梯辅助变量".内选4tag := "输入变量"."1号梯轿内选层按钮4";
   IF #_w6 AND ("一梯辅助变量".一号梯楼层数 <> 4) THEN "一梯辅助变量".一号梯内选4 := TRUE; END_IF;
   "输出变量"."1号梯4层按钮指示灯" := "一梯辅助变量".一号梯内选4;
   IF "一梯辅助变量".停在4层 AND "输出变量"."1号梯开门继电器" THEN "一梯辅助变量".一号梯内选4 := FALSE; END_IF;
   #_w7 := (("输出变量"."1号梯上行指示" AND ("一梯辅助变量".一号梯楼层数 < 5)) OR ("输出变量"."1号梯下行指示" AND ("一梯辅助变量".一号梯楼层数 > 5))) AND "输入变量"."1号梯轿内选层按钮5" AND NOT "一梯辅助变量".内选5tag;   // rising edge of "输入变量"."1号梯轿内选层按钮5"
   "一梯辅助变量".内选5tag := "输入变量"."1号梯轿内选层按钮5";
   IF #_w7 AND ("一梯辅助变量".一号梯楼层数 <> 5) THEN "一梯辅助变量".一号梯内选5 := TRUE; END_IF;
   "输出变量"."1号梯5层按钮指示灯" := "一梯辅助变量".一号梯内选5;
   IF "一梯辅助变量".停在5层 AND "输出变量"."1号梯开门继电器" THEN "一梯辅助变量".一号梯内选5 := FALSE; END_IF;
   #_w8 := "输出变量"."1号梯上行指示" AND "输入变量"."1号梯轿内选层按钮6" AND NOT "一梯辅助变量".内选6tag;   // rising edge of "输入变量"."1号梯轿内选层按钮6"
   "一梯辅助变量".内选6tag := "输入变量"."1号梯轿内选层按钮6";
   IF #_w8 AND ("一梯辅助变量".一号梯楼层数 <> 6) THEN "一梯辅助变量".一号梯内选6 := TRUE; END_IF;
   "输出变量"."1号梯6层按钮指示灯" := "一梯辅助变量".一号梯内选6;
   IF "一梯辅助变量".停在6层 AND "输出变量"."1号梯开门继电器" THEN "一梯辅助变量".一号梯内选6 := FALSE; END_IF;
   "IEC_Timer_0_DB_4".TP(IN := ("一梯辅助变量".停在6层 AND "一梯辅助变量".上行接触器1到0) OR ("一梯辅助变量".停在1层 AND "一梯辅助变量".下行接触器1到0),
                         PT := T#100ms);
   IF "IEC_Timer_0_DB_4".Q AND "一梯辅助变量".一号梯内选1 THEN "一梯辅助变量".一号梯内选1 := FALSE; END_IF;
   IF "IEC_Timer_0_DB_4".Q AND "一梯辅助变量".一号梯内选2 THEN "一梯辅助变量".一号梯内选2 := FALSE; END_IF;
   IF "IEC_Timer_0_DB_4".Q AND "一梯辅助变量".一号梯内选3 THEN "一梯辅助变量".一号梯内选3 := FALSE; END_IF;
   IF "IEC_Timer_0_DB_4".Q AND "一梯辅助变量".一号梯内选4 THEN "一梯辅助变量".一号梯内选4 := FALSE; END_IF;
   IF "IEC_Timer_0_DB_4".Q AND "一梯辅助变量".一号梯内选5 THEN "一梯辅助变量".一号梯内选5 := FALSE; END_IF;
   IF "IEC_Timer_0_DB_4".Q AND "一梯辅助变量".一号梯内选6 THEN "一梯辅助变量".一号梯内选6 := FALSE; END_IF;
END_REGION
END_FUNCTION

FUNCTION "停层开关门" : Void   // FC3, LAD
{ S7_Optimized_Access := 'TRUE' }
VERSION : 0.1
   VAR_TEMP   // added for the SCL form of the ladder/FBD networks
      _w1 : Bool;
      _w2 : Bool;
      _w3 : Bool;
      _w4 : Bool;
      _w5 : Bool;
      _w6 : Bool;
      _w7 : Bool;
      _w8 : Bool;
      _w9 : Bool;
      _w10 : Bool;
      _w11 : Bool;
   END_VAR
BEGIN

REGION Network 1: 停层信号
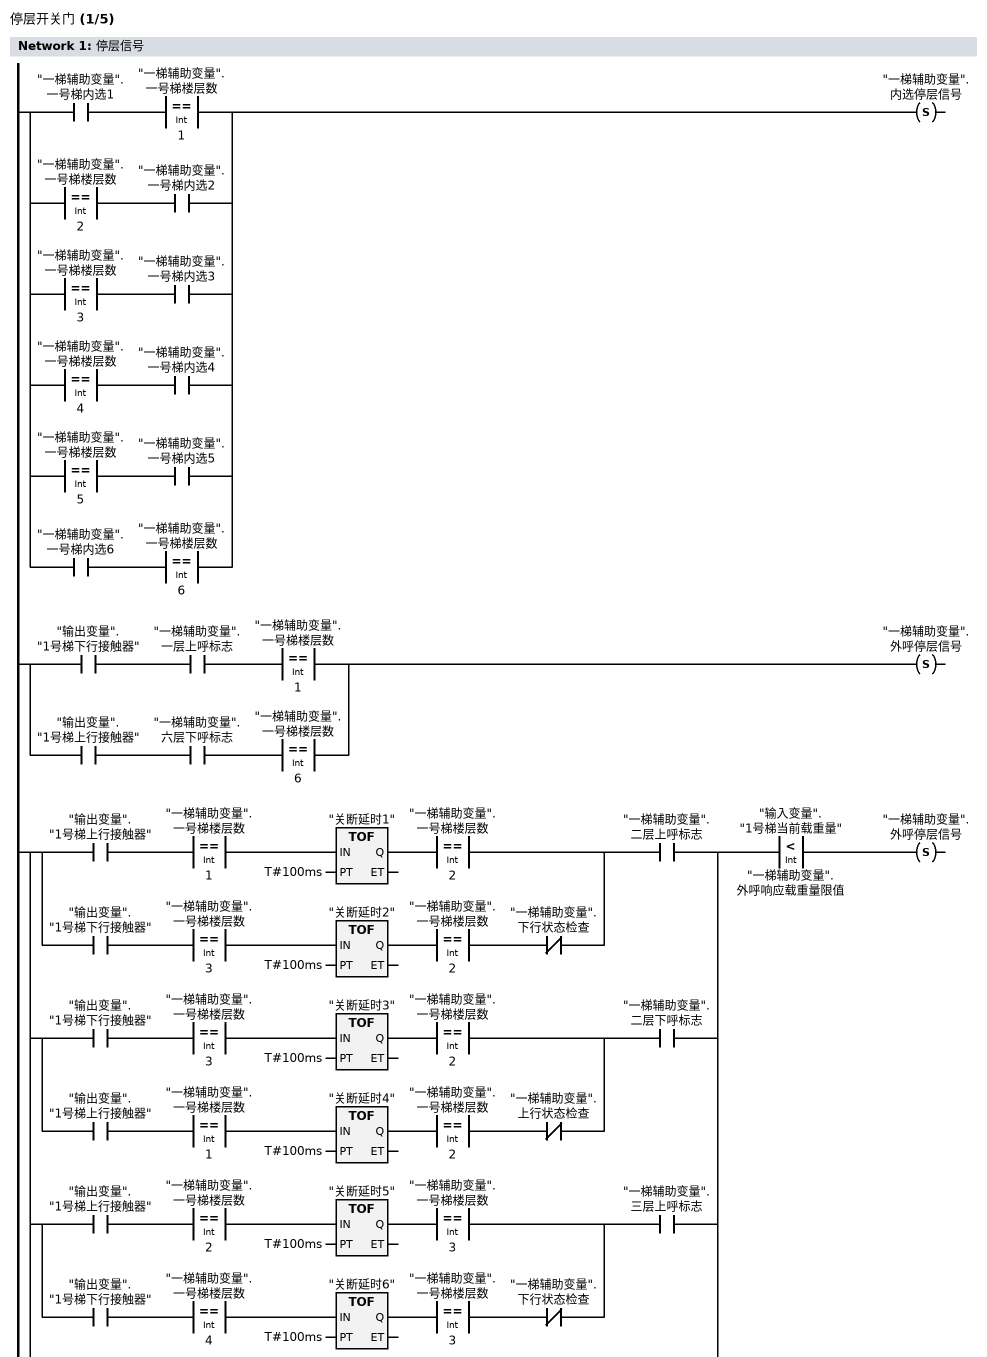
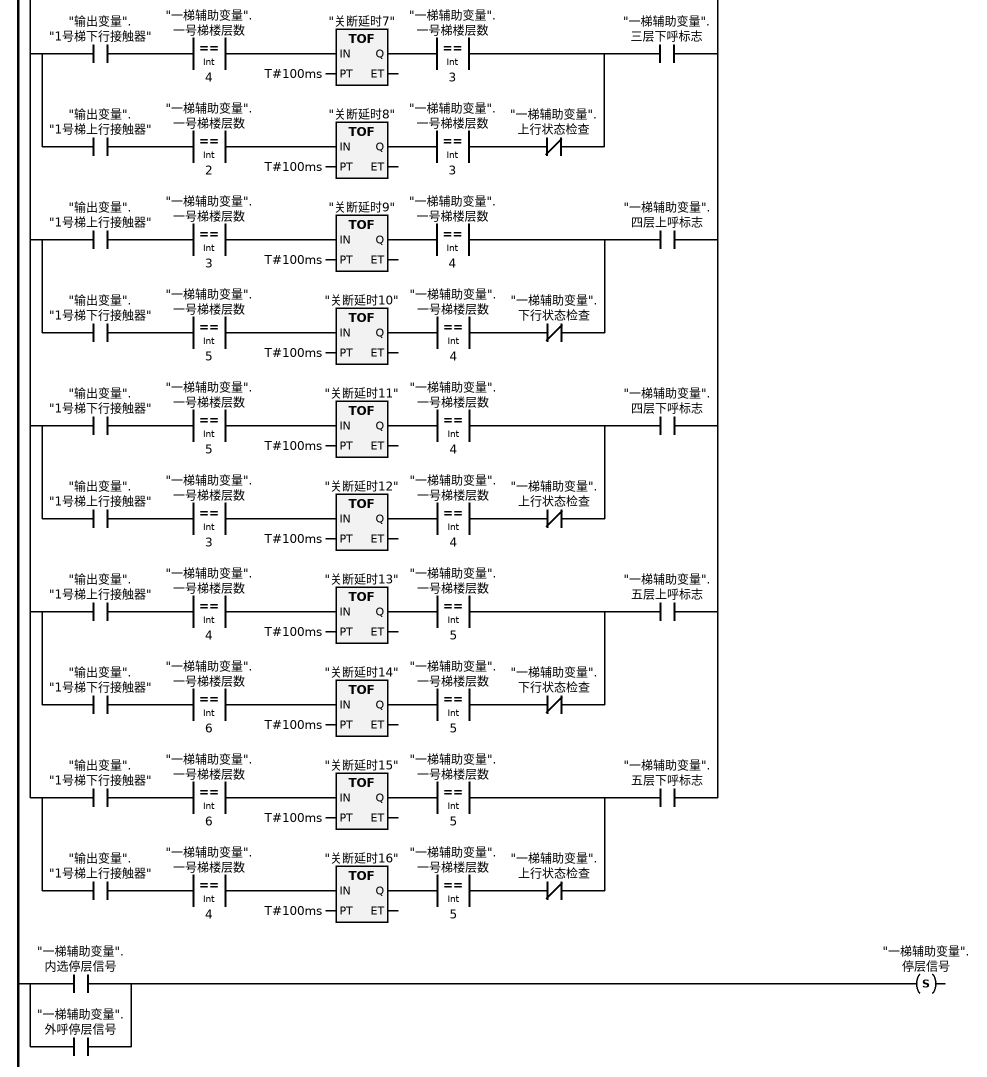
   IF ("一梯辅助变量".一号梯内选1 AND ("一梯辅助变量".一号梯楼层数 = 1)) OR (("一梯辅助变量".一号梯楼层数 = 2) AND "一梯辅助变量".一号梯内选2) OR (("一梯辅助变量".一号梯楼层数 = 3) AND "一梯辅助变量".一号梯内选3) OR (("一梯辅助变量".一号梯楼层数 = 4) AND "一梯辅助变量".一号梯内选4) OR (("一梯辅助变量".一号梯楼层数 = 5) AND "一梯辅助变量".一号梯内选5) OR ("一梯辅助变量".一号梯内选6 AND ("一梯辅助变量".一号梯楼层数 = 6)) THEN
       "一梯辅助变量".内选停层信号 := TRUE;
   END_IF;
   IF ("输出变量"."1号梯下行接触器" AND "一梯辅助变量".一层上呼标志 AND ("一梯辅助变量".一号梯楼层数 = 1)) OR ("输出变量"."1号梯上行接触器" AND "一梯辅助变量".六层下呼标志 AND ("一梯辅助变量".一号梯楼层数 = 6)) THEN
       "一梯辅助变量".外呼停层信号 := TRUE;
   END_IF;
   "关断延时1".TOF(IN := "输出变量"."1号梯上行接触器" AND ("一梯辅助变量".一号梯楼层数 = 1), PT := T#100ms);
   "关断延时2".TOF(IN := "输出变量"."1号梯下行接触器" AND ("一梯辅助变量".一号梯楼层数 = 3), PT := T#100ms);
   "关断延时3".TOF(IN := "输出变量"."1号梯下行接触器" AND ("一梯辅助变量".一号梯楼层数 = 3), PT := T#100ms);
   "关断延时4".TOF(IN := "输出变量"."1号梯上行接触器" AND ("一梯辅助变量".一号梯楼层数 = 1), PT := T#100ms);
   "关断延时5".TOF(IN := "输出变量"."1号梯上行接触器" AND ("一梯辅助变量".一号梯楼层数 = 2), PT := T#100ms);
   "关断延时6".TOF(IN := "输出变量"."1号梯下行接触器" AND ("一梯辅助变量".一号梯楼层数 = 4), PT := T#100ms);
   "关断延时7".TOF(IN := "输出变量"."1号梯下行接触器" AND ("一梯辅助变量".一号梯楼层数 = 4), PT := T#100ms);
   "关断延时8".TOF(IN := "输出变量"."1号梯上行接触器" AND ("一梯辅助变量".一号梯楼层数 = 2), PT := T#100ms);
   "关断延时9".TOF(IN := "输出变量"."1号梯上行接触器" AND ("一梯辅助变量".一号梯楼层数 = 3), PT := T#100ms);
   "关断延时10".TOF(IN := "输出变量"."1号梯下行接触器" AND ("一梯辅助变量".一号梯楼层数 = 5), PT := T#100ms);
   "关断延时11".TOF(IN := "输出变量"."1号梯下行接触器" AND ("一梯辅助变量".一号梯楼层数 = 5), PT := T#100ms);
   "关断延时12".TOF(IN := "输出变量"."1号梯上行接触器" AND ("一梯辅助变量".一号梯楼层数 = 3), PT := T#100ms);
   "关断延时13".TOF(IN := "输出变量"."1号梯上行接触器" AND ("一梯辅助变量".一号梯楼层数 = 4), PT := T#100ms);
   "关断延时14".TOF(IN := "输出变量"."1号梯下行接触器" AND ("一梯辅助变量".一号梯楼层数 = 6), PT := T#100ms);
   "关断延时15".TOF(IN := "输出变量"."1号梯下行接触器" AND ("一梯辅助变量".一号梯楼层数 = 6), PT := T#100ms);
   "关断延时16".TOF(IN := "输出变量"."1号梯上行接触器" AND ("一梯辅助变量".一号梯楼层数 = 4), PT := T#100ms);
   IF (((("关断延时1".Q AND ("一梯辅助变量".一号梯楼层数 = 2)) OR ("关断延时2".Q AND ("一梯辅助变量".一号梯楼层数 = 2) AND NOT "一梯辅助变量".下行状态检查)) AND "一梯辅助变量".二层上呼标志) OR ((("关断延时3".Q AND ("一梯辅助变量".一号梯楼层数 = 2)) OR ("关断延时4".Q AND ("一梯辅助变量".一号梯楼层数 = 2) AND NOT "一梯辅助变量".上行状态检查)) AND "一梯辅助变量".二层下呼标志) OR ((("关断延时5".Q AND ("一梯辅助变量".一号梯楼层数 = 3)) OR ("关断延时6".Q AND ("一梯辅助变量".一号梯楼层数 = 3) AND NOT "一梯辅助变量".下行状态检查)) AND "一梯辅助变量".三层上呼标志) OR ((("关断延时7".Q AND ("一梯辅助变量".一号梯楼层数 = 3)) OR ("关断延时8".Q AND ("一梯辅助变量".一号梯楼层数 = 3) AND NOT "一梯辅助变量".上行状态检查)) AND "一梯辅助变量".三层下呼标志) OR ((("关断延时9".Q AND ("一梯辅助变量".一号梯楼层数 = 4)) OR ("关断延时10".Q AND ("一梯辅助变量".一号梯楼层数 = 4) AND NOT "一梯辅助变量".下行状态检查)) AND "一梯辅助变量".四层上呼标志) OR ((("关断延时11".Q AND ("一梯辅助变量".一号梯楼层数 = 4)) OR ("关断延时12".Q AND ("一梯辅助变量".一号梯楼层数 = 4) AND NOT "一梯辅助变量".上行状态检查)) AND "一梯辅助变量".四层下呼标志) OR ((("关断延时13".Q AND ("一梯辅助变量".一号梯楼层数 = 5)) OR ("关断延时14".Q AND ("一梯辅助变量".一号梯楼层数 = 5) AND NOT "一梯辅助变量".下行状态检查)) AND "一梯辅助变量".五层上呼标志) OR ((("关断延时15".Q AND ("一梯辅助变量".一号梯楼层数 = 5)) OR ("关断延时16".Q AND ("一梯辅助变量".一号梯楼层数 = 5) AND NOT "一梯辅助变量".上行状态检查)) AND "一梯辅助变量".五层下呼标志)) AND ("输入变量"."1号梯当前载重量" < "一梯辅助变量".外呼响应载重量限值) THEN
       "一梯辅助变量".外呼停层信号 := TRUE;
   END_IF;
   IF "一梯辅助变量".内选停层信号 OR "一梯辅助变量".外呼停层信号 THEN "一梯辅助变量".停层信号 := TRUE; END_IF;
END_REGION

REGION Network 2: 准备停层，三级减速到指定位置
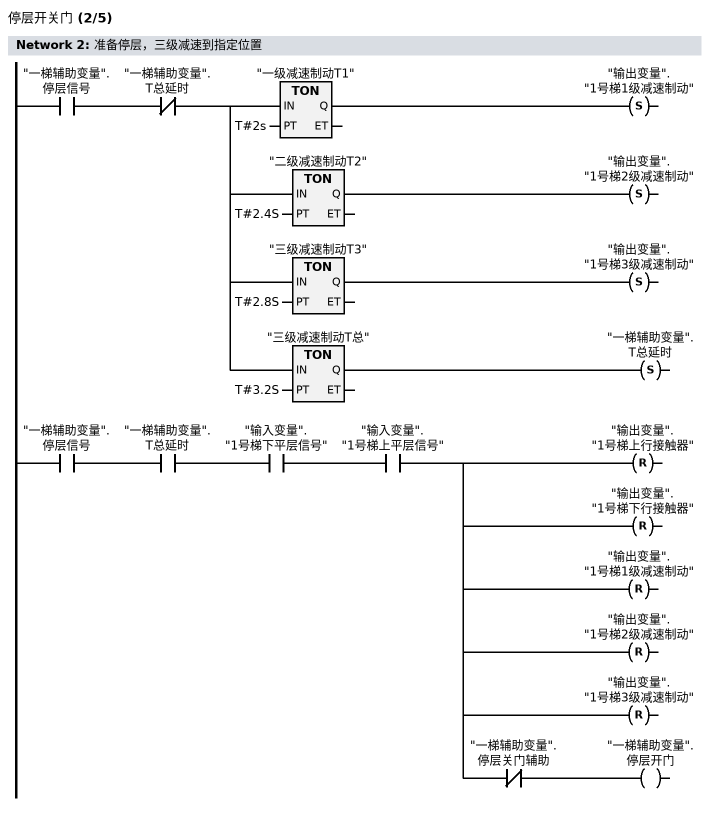
   #_w1 := "一梯辅助变量".停层信号 AND NOT "一梯辅助变量".T总延时;
   "一级减速制动T1".TON(IN := #_w1, PT := T#2s);
   IF "一级减速制动T1".Q THEN "输出变量"."1号梯1级减速制动" := TRUE; END_IF;
   "二级减速制动T2".TON(IN := #_w1, PT := T#2.4S);
   IF "二级减速制动T2".Q THEN "输出变量"."1号梯2级减速制动" := TRUE; END_IF;
   "三级减速制动T3".TON(IN := #_w1, PT := T#2.8S);
   IF "三级减速制动T3".Q THEN "输出变量"."1号梯3级减速制动" := TRUE; END_IF;
   "三级减速制动T总".TON(IN := #_w1, PT := T#3.2S);
   IF "三级减速制动T总".Q THEN "一梯辅助变量".T总延时 := TRUE; END_IF;
   #_w2 := "一梯辅助变量".停层信号 AND "一梯辅助变量".T总延时 AND "输入变量"."1号梯下平层信号" AND "输入变量"."1号梯上平层信号";
   IF #_w2 THEN
       "输出变量"."1号梯上行接触器" := FALSE;
       "输出变量"."1号梯下行接触器" := FALSE;
       "输出变量"."1号梯1级减速制动" := FALSE;
       "输出变量"."1号梯2级减速制动" := FALSE;
       "输出变量"."1号梯3级减速制动" := FALSE;
   END_IF;
   "一梯辅助变量".停层开门 := #_w2 AND NOT "一梯辅助变量".停层关门辅助;
END_REGION

REGION Network 3: 开关门（停层、开门按钮、本层上下呼、光幕、超重）
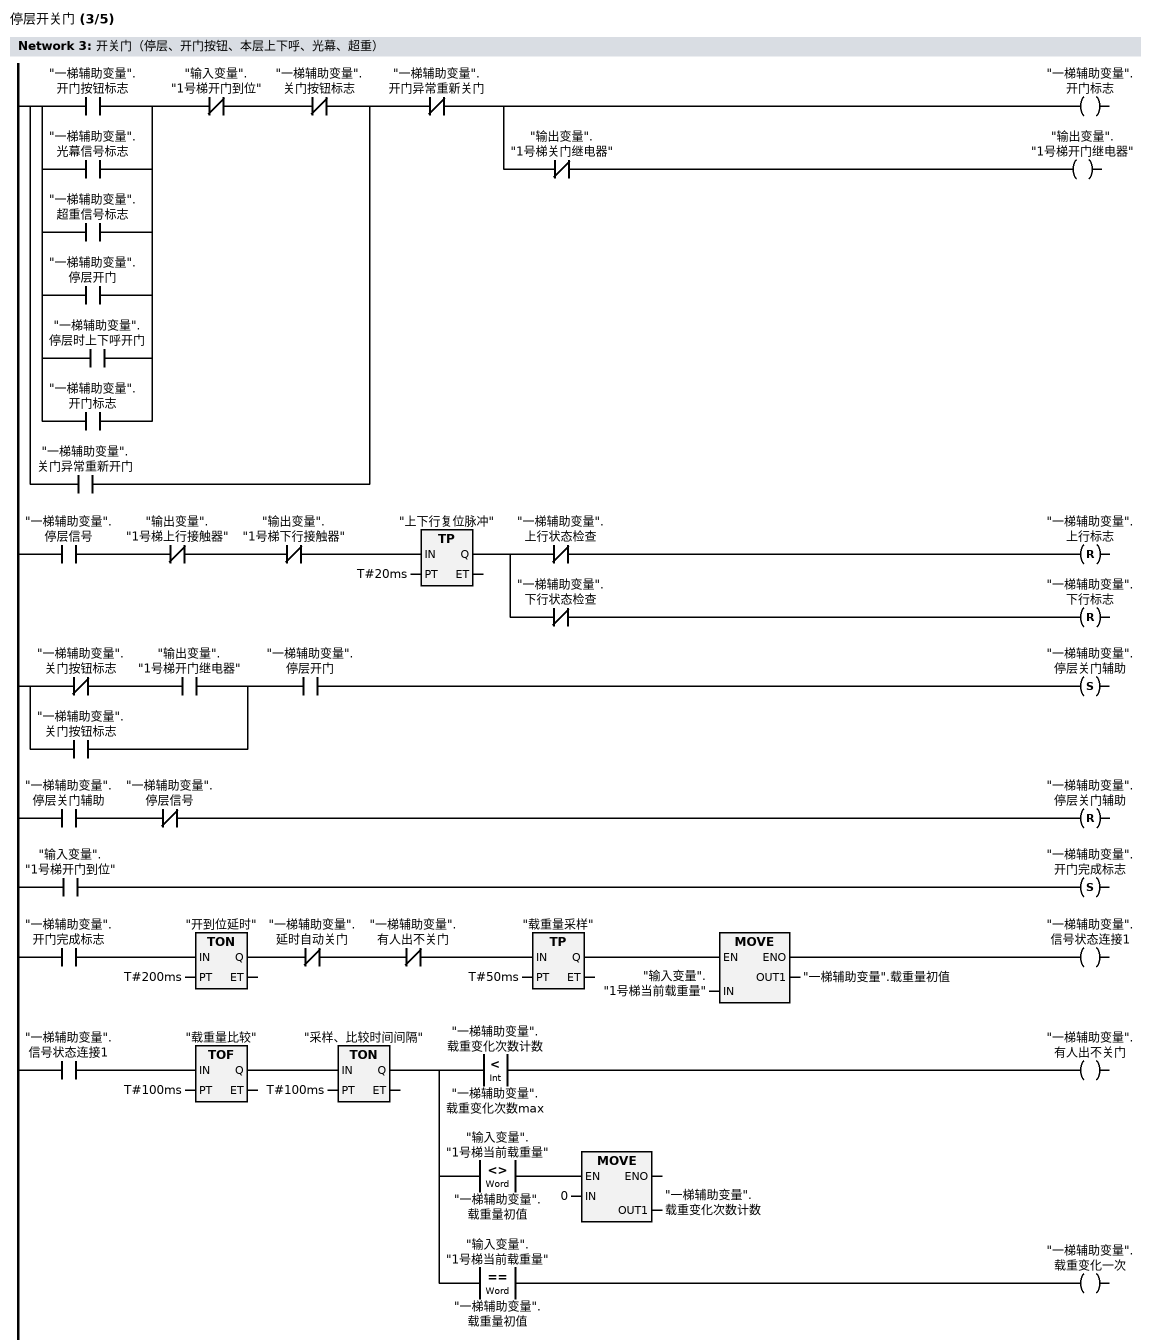
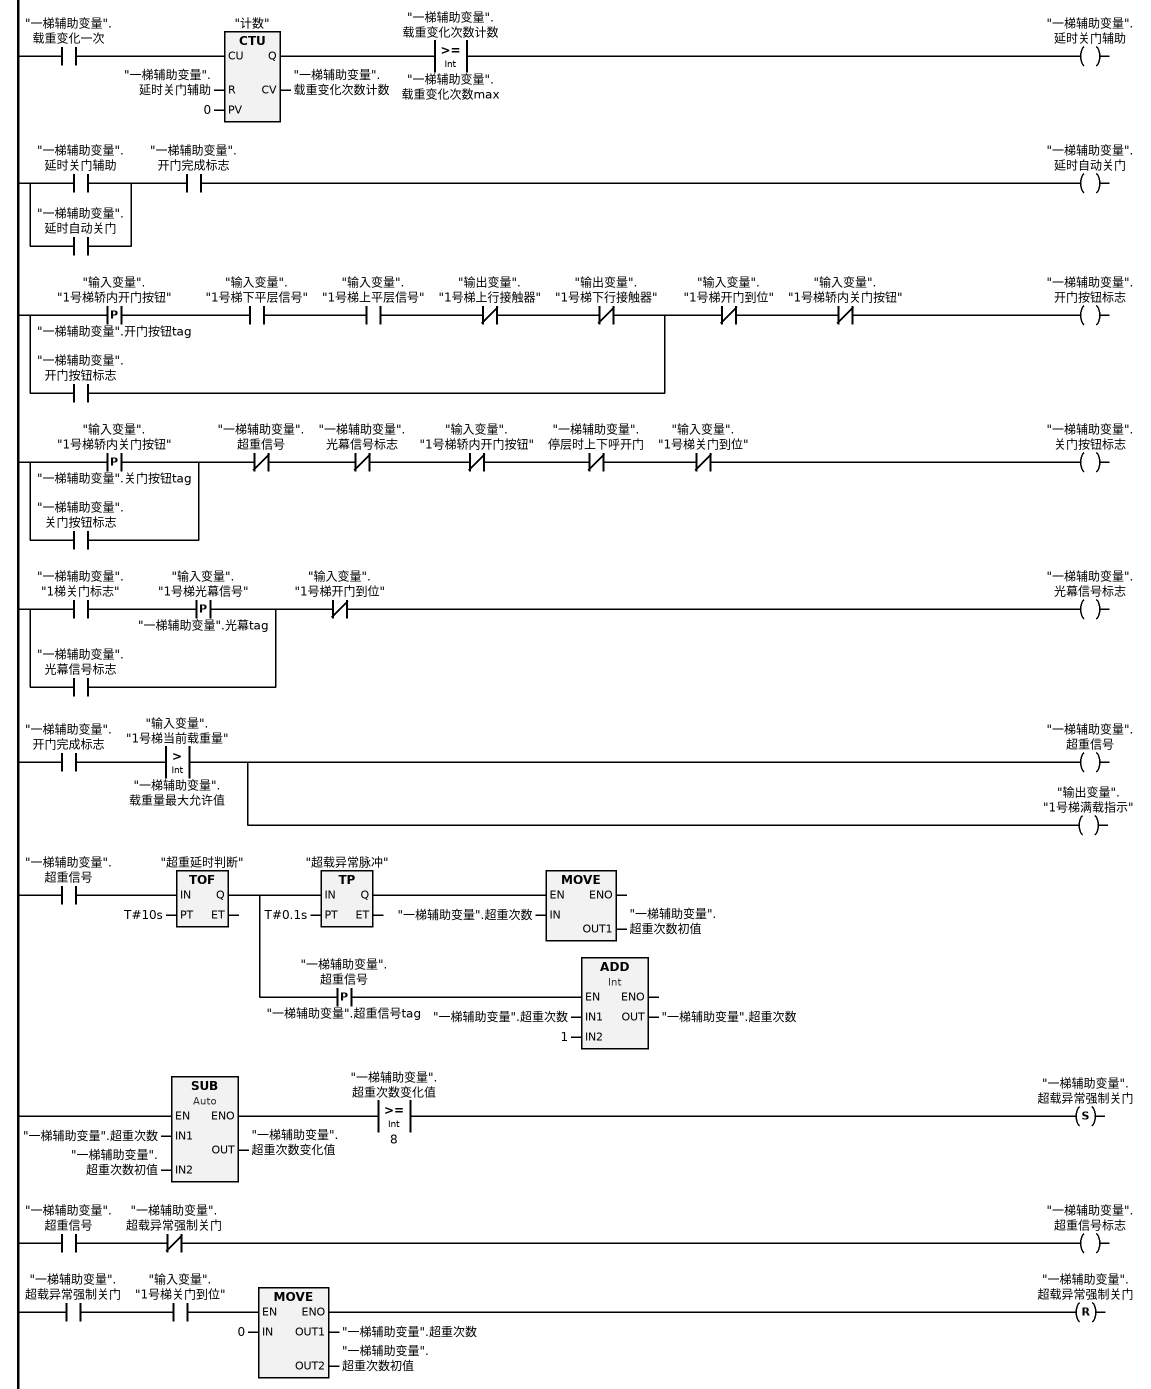
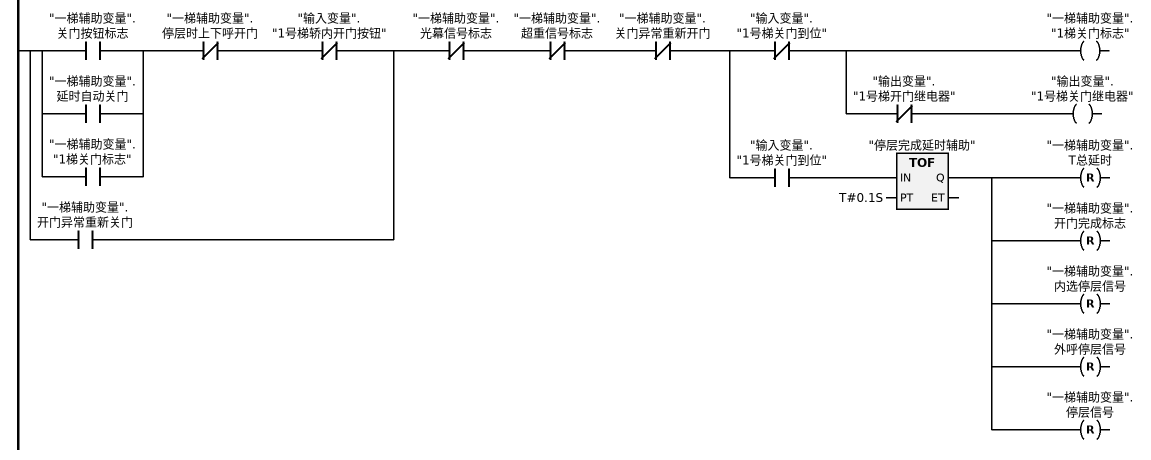
   "一梯辅助变量".开门标志 := ((("一梯辅助变量".开门按钮标志 OR "一梯辅助变量".光幕信号标志 OR "一梯辅助变量".超重信号标志 OR "一梯辅助变量".停层开门 OR "一梯辅助变量".停层时上下呼开门 OR "一梯辅助变量".开门标志) AND NOT "输入变量"."1号梯开门到位" AND NOT "一梯辅助变量".关门按钮标志) OR "一梯辅助变量".关门异常重新开门) AND NOT "一梯辅助变量".开门异常重新关门;
   "输出变量"."1号梯开门继电器" := "一梯辅助变量".开门标志 AND NOT "输出变量"."1号梯关门继电器";
   "上下行复位脉冲".TP(IN := "一梯辅助变量".停层信号 AND NOT "输出变量"."1号梯上行接触器" AND NOT "输出变量"."1号梯下行接触器", PT := T#20ms);
   IF "上下行复位脉冲".Q AND NOT "一梯辅助变量".上行状态检查 THEN "一梯辅助变量".上行标志 := FALSE; END_IF;
   IF "上下行复位脉冲".Q AND NOT "一梯辅助变量".下行状态检查 THEN "一梯辅助变量".下行标志 := FALSE; END_IF;
   IF ((NOT "一梯辅助变量".关门按钮标志 AND "输出变量"."1号梯开门继电器") OR "一梯辅助变量".关门按钮标志) AND "一梯辅助变量".停层开门 THEN
       "一梯辅助变量".停层关门辅助 := TRUE;
   END_IF;
   IF "一梯辅助变量".停层关门辅助 AND NOT "一梯辅助变量".停层信号 THEN "一梯辅助变量".停层关门辅助 := FALSE; END_IF;
   IF "输入变量"."1号梯开门到位" THEN "一梯辅助变量".开门完成标志 := TRUE; END_IF;
   "开到位延时".TON(IN := "一梯辅助变量".开门完成标志, PT := T#200ms);
   "载重量采样".TP(IN := "开到位延时".Q AND NOT "一梯辅助变量".延时自动关门 AND NOT "一梯辅助变量".有人出不关门, PT := T#50ms);
   IF "载重量采样".Q THEN "一梯辅助变量".载重量初值 := "输入变量"."1号梯当前载重量"; END_IF;
   "一梯辅助变量".信号状态连接1 := "载重量采样".Q;
   "载重量比较".TOF(IN := "一梯辅助变量".信号状态连接1, PT := T#100ms);
   "采样、比较时间间隔".TON(IN := "载重量比较".Q, PT := T#100ms);
   "一梯辅助变量".有人出不关门 := "采样、比较时间间隔".Q AND ("一梯辅助变量".载重变化次数计数 < "一梯辅助变量".载重变化次数max);
   IF "采样、比较时间间隔".Q AND ("输入变量"."1号梯当前载重量" <> "一梯辅助变量".载重量初值) THEN "一梯辅助变量".载重变化次数计数 := 0; END_IF;
   "一梯辅助变量".载重变化一次 := "采样、比较时间间隔".Q AND ("输入变量"."1号梯当前载重量" = "一梯辅助变量".载重量初值);
   "计数".CTU(CU := "一梯辅助变量".载重变化一次, R := "一梯辅助变量".延时关门辅助, PV := 0, CV => "一梯辅助变量".载重变化次数计数);
   "一梯辅助变量".延时关门辅助 := "计数".Q AND ("一梯辅助变量".载重变化次数计数 >= "一梯辅助变量".载重变化次数max);
   "一梯辅助变量".延时自动关门 := ("一梯辅助变量".延时关门辅助 OR "一梯辅助变量".延时自动关门) AND "一梯辅助变量".开门完成标志;
   #_w1 := "输入变量"."1号梯轿内开门按钮" AND NOT "一梯辅助变量".开门按钮tag;   // rising edge of "输入变量"."1号梯轿内开门按钮"
   "一梯辅助变量".开门按钮tag := "输入变量"."1号梯轿内开门按钮";
   "一梯辅助变量".开门按钮标志 := ((#_w1 AND "输入变量"."1号梯下平层信号" AND "输入变量"."1号梯上平层信号" AND NOT "输出变量"."1号梯上行接触器" AND NOT "输出变量"."1号梯下行接触器") OR "一梯辅助变量".开门按钮标志) AND NOT "输入变量"."1号梯开门到位" AND NOT "输入变量"."1号梯轿内关门按钮";
   #_w2 := "输入变量"."1号梯轿内关门按钮" AND NOT "一梯辅助变量".关门按钮tag;   // rising edge of "输入变量"."1号梯轿内关门按钮"
   "一梯辅助变量".关门按钮tag := "输入变量"."1号梯轿内关门按钮";
   "一梯辅助变量".关门按钮标志 := (#_w2 OR "一梯辅助变量".关门按钮标志) AND NOT "一梯辅助变量".超重信号 AND NOT "一梯辅助变量".光幕信号标志 AND NOT "输入变量"."1号梯轿内开门按钮" AND NOT "一梯辅助变量".停层时上下呼开门 AND NOT "输入变量"."1号梯关门到位";
   #_w3 := "一梯辅助变量"."1梯关门标志" AND "输入变量"."1号梯光幕信号" AND NOT "一梯辅助变量".光幕tag;   // rising edge of "输入变量"."1号梯光幕信号"
   "一梯辅助变量".光幕tag := "输入变量"."1号梯光幕信号";
   "一梯辅助变量".光幕信号标志 := (#_w3 OR "一梯辅助变量".光幕信号标志) AND NOT "输入变量"."1号梯开门到位";
   "一梯辅助变量".超重信号 := "一梯辅助变量".开门完成标志 AND ("输入变量"."1号梯当前载重量" > "一梯辅助变量".载重量最大允许值);
   "输出变量"."1号梯满载指示" := "一梯辅助变量".超重信号;
   "超重延时判断".TOF(IN := "一梯辅助变量".超重信号, PT := T#10s);
   "超载异常脉冲".TP(IN := "超重延时判断".Q, PT := T#0.1s);
   IF "超载异常脉冲".Q THEN "一梯辅助变量".超重次数初值 := "一梯辅助变量".超重次数; END_IF;
   #_w4 := "超重延时判断".Q AND "一梯辅助变量".超重信号 AND NOT "一梯辅助变量".超重信号tag;   // rising edge of "一梯辅助变量".超重信号
   "一梯辅助变量".超重信号tag := "一梯辅助变量".超重信号;
   IF #_w4 THEN "一梯辅助变量".超重次数 := "一梯辅助变量".超重次数 + 1; END_IF;
   "一梯辅助变量".超重次数变化值 := "一梯辅助变量".超重次数 - "一梯辅助变量".超重次数初值;
   IF "一梯辅助变量".超重次数变化值 >= 8 THEN "一梯辅助变量".超载异常强制关门 := TRUE; END_IF;
   "一梯辅助变量".超重信号标志 := "一梯辅助变量".超重信号 AND NOT "一梯辅助变量".超载异常强制关门;
   IF "一梯辅助变量".超载异常强制关门 AND "输入变量"."1号梯关门到位" THEN
       "一梯辅助变量".超重次数 := 0;
       "一梯辅助变量".超重次数初值 := 0;
       "一梯辅助变量".超载异常强制关门 := FALSE;
   END_IF;
   #_w5 := ((("一梯辅助变量".关门按钮标志 OR "一梯辅助变量".延时自动关门 OR "一梯辅助变量"."1梯关门标志") AND NOT "一梯辅助变量".停层时上下呼开门 AND NOT "输入变量"."1号梯轿内开门按钮") OR "一梯辅助变量".开门异常重新关门) AND NOT "一梯辅助变量".光幕信号标志 AND NOT "一梯辅助变量".超重信号标志 AND NOT "一梯辅助变量".关门异常重新开门;
   "一梯辅助变量"."1梯关门标志" := #_w5 AND NOT "输入变量"."1号梯关门到位";
   "输出变量"."1号梯关门继电器" := "一梯辅助变量"."1梯关门标志" AND NOT "输出变量"."1号梯开门继电器";
   "停层完成延时辅助".TOF(IN := #_w5 AND "输入变量"."1号梯关门到位", PT := T#0.1S);
   IF "停层完成延时辅助".Q THEN
       "一梯辅助变量".T总延时 := FALSE;
       "一梯辅助变量".开门完成标志 := FALSE;
       "一梯辅助变量".内选停层信号 := FALSE;
       "一梯辅助变量".外呼停层信号 := FALSE;
       "一梯辅助变量".停层信号 := FALSE;
   END_IF;
END_REGION

REGION Network 4: 本层的上下呼梯开关门
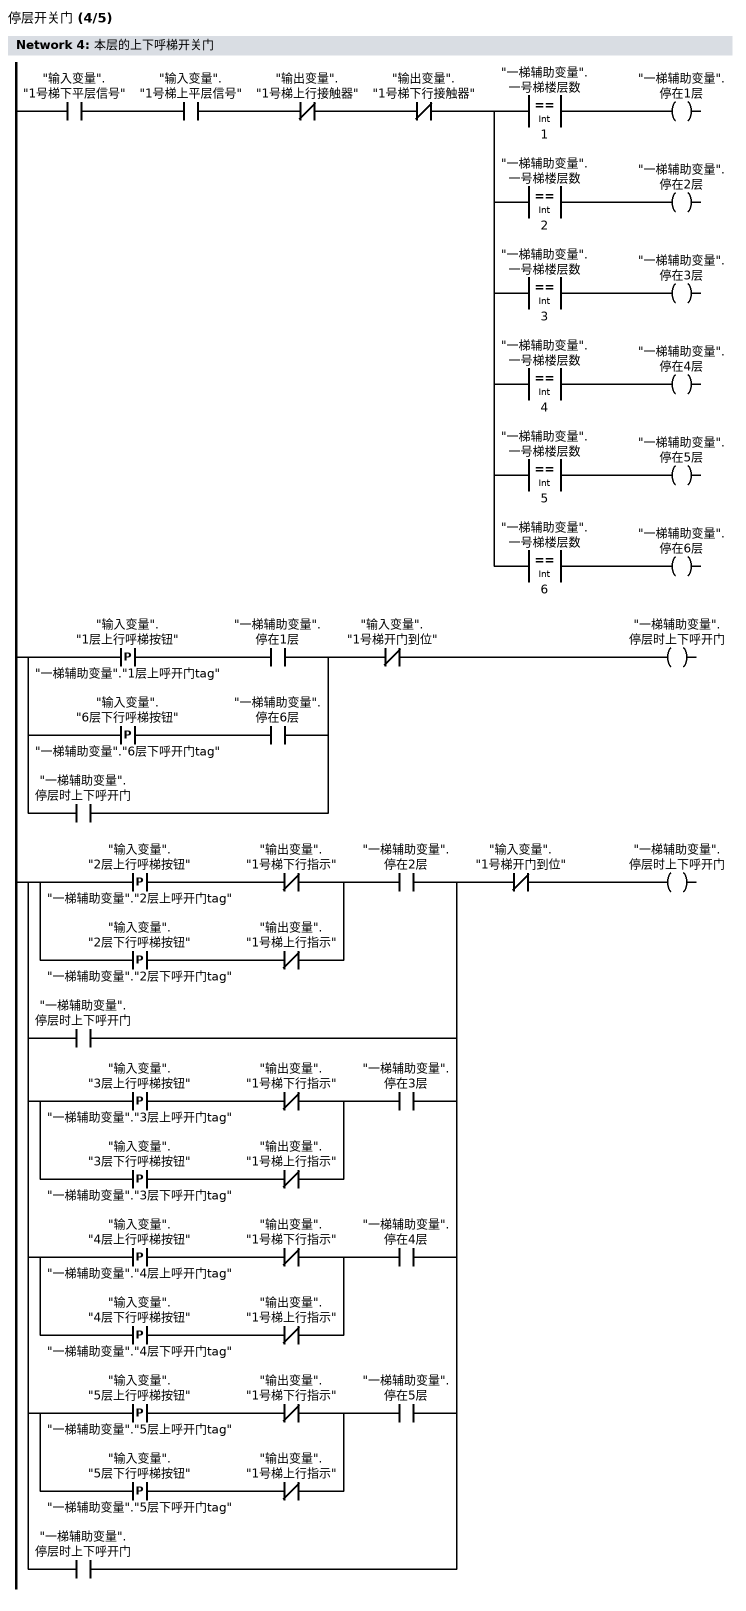
   RUNG wire#powerrail
      Contact( "输入变量"."1号梯下平层信号" )
      Contact( "输入变量"."1号梯上平层信号" )
      I_Contact( "输出变量"."1号梯上行接触器" )
      I_Contact( "输出变量"."1号梯下行接触器" )
      wire#w1
      { S7_Templates := "SrcType := Int" } EQ_Contact(in1 := "一梯辅助变量".一号梯楼层数, in2 := 1)
      Coil( "一梯辅助变量".停在1层 )
   END_RUNG
   RUNG wire#w1
      { S7_Templates := "SrcType := Int" } EQ_Contact(in1 := "一梯辅助变量".一号梯楼层数, in2 := 2)
      Coil( "一梯辅助变量".停在2层 )
   END_RUNG
   RUNG wire#w1
      { S7_Templates := "SrcType := Int" } EQ_Contact(in1 := "一梯辅助变量".一号梯楼层数, in2 := 3)
      Coil( "一梯辅助变量".停在3层 )
   END_RUNG
   RUNG wire#w1
      { S7_Templates := "SrcType := Int" } EQ_Contact(in1 := "一梯辅助变量".一号梯楼层数, in2 := 4)
      Coil( "一梯辅助变量".停在4层 )
   END_RUNG
   RUNG wire#w1
      { S7_Templates := "SrcType := Int" } EQ_Contact(in1 := "一梯辅助变量".一号梯楼层数, in2 := 5)
      Coil( "一梯辅助变量".停在5层 )
   END_RUNG
   RUNG wire#w1
      { S7_Templates := "SrcType := Int" } EQ_Contact(in1 := "一梯辅助变量".一号梯楼层数, in2 := 6)
      Coil( "一梯辅助变量".停在6层 )
   END_RUNG
   RUNG wire#powerrail
      P_Contact(operand := "输入变量"."1层上行呼梯按钮", bit := "一梯辅助变量"."1层上呼开门tag")
      Contact( "一梯辅助变量".停在1层 )
      wire#w2
      I_Contact( "输入变量"."1号梯开门到位" )
      Coil( "一梯辅助变量".停层时上下呼开门 )
   END_RUNG
   RUNG wire#powerrail
      P_Contact(operand := "输入变量"."6层下行呼梯按钮", bit := "一梯辅助变量"."6层下呼开门tag")
      Contact( "一梯辅助变量".停在6层 )
   END_RUNG wire#w2
   RUNG wire#powerrail
      Contact( "一梯辅助变量".停层时上下呼开门 )
   END_RUNG wire#w2
   RUNG wire#powerrail
      P_Contact(operand := "输入变量"."2层上行呼梯按钮", bit := "一梯辅助变量"."2层上呼开门tag")
      I_Contact( "输出变量"."1号梯下行指示" )
      wire#w3
      Contact( "一梯辅助变量".停在2层 )
      wire#w4
      I_Contact( "输入变量"."1号梯开门到位" )
      Coil( "一梯辅助变量".停层时上下呼开门 )
   END_RUNG
   RUNG wire#powerrail
      P_Contact(operand := "输入变量"."2层下行呼梯按钮", bit := "一梯辅助变量"."2层下呼开门tag")
      I_Contact( "输出变量"."1号梯上行指示" )
   END_RUNG wire#w3
   RUNG wire#powerrail
      Contact( "一梯辅助变量".停层时上下呼开门 )
   END_RUNG wire#w4
   RUNG wire#powerrail
      P_Contact(operand := "输入变量"."3层上行呼梯按钮", bit := "一梯辅助变量"."3层上呼开门tag")
      I_Contact( "输出变量"."1号梯下行指示" )
      wire#w5
      Contact( "一梯辅助变量".停在3层 )
   END_RUNG wire#w4
   RUNG wire#powerrail
      P_Contact(operand := "输入变量"."3层下行呼梯按钮", bit := "一梯辅助变量"."3层下呼开门tag")
      I_Contact( "输出变量"."1号梯上行指示" )
   END_RUNG wire#w5
   RUNG wire#powerrail
      P_Contact(operand := "输入变量"."4层上行呼梯按钮", bit := "一梯辅助变量"."4层上呼开门tag")
      I_Contact( "输出变量"."1号梯下行指示" )
      wire#w6
      Contact( "一梯辅助变量".停在4层 )
   END_RUNG wire#w4
   RUNG wire#powerrail
      P_Contact(operand := "输入变量"."4层下行呼梯按钮", bit := "一梯辅助变量"."4层下呼开门tag")
      I_Contact( "输出变量"."1号梯上行指示" )
   END_RUNG wire#w6
   RUNG wire#powerrail
      P_Contact(operand := "输入变量"."5层上行呼梯按钮", bit := "一梯辅助变量"."5层上呼开门tag")
      I_Contact( "输出变量"."1号梯下行指示" )
      wire#w7
      Contact( "一梯辅助变量".停在5层 )
   END_RUNG wire#w4
   RUNG wire#powerrail
      P_Contact(operand := "输入变量"."5层下行呼梯按钮", bit := "一梯辅助变量"."5层下呼开门tag")
      I_Contact( "输出变量"."1号梯上行指示" )
   END_RUNG wire#w7
   RUNG wire#powerrail
      Contact( "一梯辅助变量".停层时上下呼开门 )
   END_RUNG wire#w4
   // the same network as SCL:
   #_w1 := "输入变量"."1号梯下平层信号" AND "输入变量"."1号梯上平层信号" AND NOT "输出变量"."1号梯上行接触器" AND NOT "输出变量"."1号梯下行接触器";
   "一梯辅助变量".停在1层 := #_w1 AND ("一梯辅助变量".一号梯楼层数 = 1);
   "一梯辅助变量".停在2层 := #_w1 AND ("一梯辅助变量".一号梯楼层数 = 2);
   "一梯辅助变量".停在3层 := #_w1 AND ("一梯辅助变量".一号梯楼层数 = 3);
   "一梯辅助变量".停在4层 := #_w1 AND ("一梯辅助变量".一号梯楼层数 = 4);
   "一梯辅助变量".停在5层 := #_w1 AND ("一梯辅助变量".一号梯楼层数 = 5);
   "一梯辅助变量".停在6层 := #_w1 AND ("一梯辅助变量".一号梯楼层数 = 6);
   #_w2 := "输入变量"."1层上行呼梯按钮" AND NOT "一梯辅助变量"."1层上呼开门tag";   // rising edge of "输入变量"."1层上行呼梯按钮"
   "一梯辅助变量"."1层上呼开门tag" := "输入变量"."1层上行呼梯按钮";
   #_w3 := "输入变量"."6层下行呼梯按钮" AND NOT "一梯辅助变量"."6层下呼开门tag";   // rising edge of "输入变量"."6层下行呼梯按钮"
   "一梯辅助变量"."6层下呼开门tag" := "输入变量"."6层下行呼梯按钮";
   "一梯辅助变量".停层时上下呼开门 := ((#_w2 AND "一梯辅助变量".停在1层) OR (#_w3 AND "一梯辅助变量".停在6层) OR "一梯辅助变量".停层时上下呼开门) AND NOT "输入变量"."1号梯开门到位";
   #_w4 := "输入变量"."2层上行呼梯按钮" AND NOT "一梯辅助变量"."2层上呼开门tag";   // rising edge of "输入变量"."2层上行呼梯按钮"
   "一梯辅助变量"."2层上呼开门tag" := "输入变量"."2层上行呼梯按钮";
   #_w5 := "输入变量"."2层下行呼梯按钮" AND NOT "一梯辅助变量"."2层下呼开门tag";   // rising edge of "输入变量"."2层下行呼梯按钮"
   "一梯辅助变量"."2层下呼开门tag" := "输入变量"."2层下行呼梯按钮";
   #_w6 := "输入变量"."3层上行呼梯按钮" AND NOT "一梯辅助变量"."3层上呼开门tag";   // rising edge of "输入变量"."3层上行呼梯按钮"
   "一梯辅助变量"."3层上呼开门tag" := "输入变量"."3层上行呼梯按钮";
   #_w7 := "输入变量"."3层下行呼梯按钮" AND NOT "一梯辅助变量"."3层下呼开门tag";   // rising edge of "输入变量"."3层下行呼梯按钮"
   "一梯辅助变量"."3层下呼开门tag" := "输入变量"."3层下行呼梯按钮";
   #_w8 := "输入变量"."4层上行呼梯按钮" AND NOT "一梯辅助变量"."4层上呼开门tag";   // rising edge of "输入变量"."4层上行呼梯按钮"
   "一梯辅助变量"."4层上呼开门tag" := "输入变量"."4层上行呼梯按钮";
   #_w9 := "输入变量"."4层下行呼梯按钮" AND NOT "一梯辅助变量"."4层下呼开门tag";   // rising edge of "输入变量"."4层下行呼梯按钮"
   "一梯辅助变量"."4层下呼开门tag" := "输入变量"."4层下行呼梯按钮";
   #_w10 := "输入变量"."5层上行呼梯按钮" AND NOT "一梯辅助变量"."5层上呼开门tag";   // rising edge of "输入变量"."5层上行呼梯按钮"
   "一梯辅助变量"."5层上呼开门tag" := "输入变量"."5层上行呼梯按钮";
   #_w11 := "输入变量"."5层下行呼梯按钮" AND NOT "一梯辅助变量"."5层下呼开门tag";   // rising edge of "输入变量"."5层下行呼梯按钮"
   "一梯辅助变量"."5层下呼开门tag" := "输入变量"."5层下行呼梯按钮";
   "一梯辅助变量".停层时上下呼开门 := ((((#_w4 AND NOT "输出变量"."1号梯下行指示") OR (#_w5 AND NOT "输出变量"."1号梯上行指示")) AND "一梯辅助变量".停在2层) OR "一梯辅助变量".停层时上下呼开门 OR (((#_w6 AND NOT "输出变量"."1号梯下行指示") OR (#_w7 AND NOT "输出变量"."1号梯上行指示")) AND "一梯辅助变量".停在3层) OR (((#_w8 AND NOT "输出变量"."1号梯下行指示") OR (#_w9 AND NOT "输出变量"."1号梯上行指示")) AND "一梯辅助变量".停在4层) OR (((#_w10 AND NOT "输出变量"."1号梯下行指示") OR (#_w11 AND NOT "输出变量"."1号梯上行指示")) AND "一梯辅助变量".停在5层) OR "一梯辅助变量".停层时上下呼开门) AND NOT "输入变量"."1号梯开门到位";
END_REGION

REGION Network 5: 高低速接触器
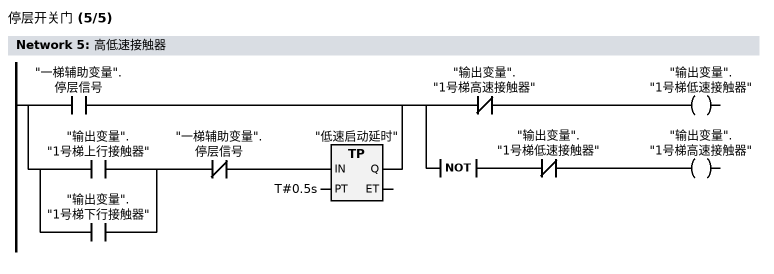
   "低速启动延时".TP(IN := ("输出变量"."1号梯上行接触器" OR "输出变量"."1号梯下行接触器") AND NOT "一梯辅助变量".停层信号, PT := T#0.5s);
   #_w1 := "一梯辅助变量".停层信号 OR "低速启动延时".Q;
   "输出变量"."1号梯低速接触器" := #_w1 AND NOT "输出变量"."1号梯高速接触器";
   "输出变量"."1号梯高速接触器" := NOT #_w1 AND NOT "输出变量"."1号梯低速接触器";
END_REGION
END_FUNCTION

FUNCTION "其它" : Void   // FC4, LAD
{ S7_Optimized_Access := 'TRUE' }
VERSION : 0.1
   VAR_TEMP   // added for the SCL form of the ladder/FBD networks
      _w1 : Bool;
      _w2 : Bool;
   END_VAR
BEGIN

REGION Network 1: 待载休眠
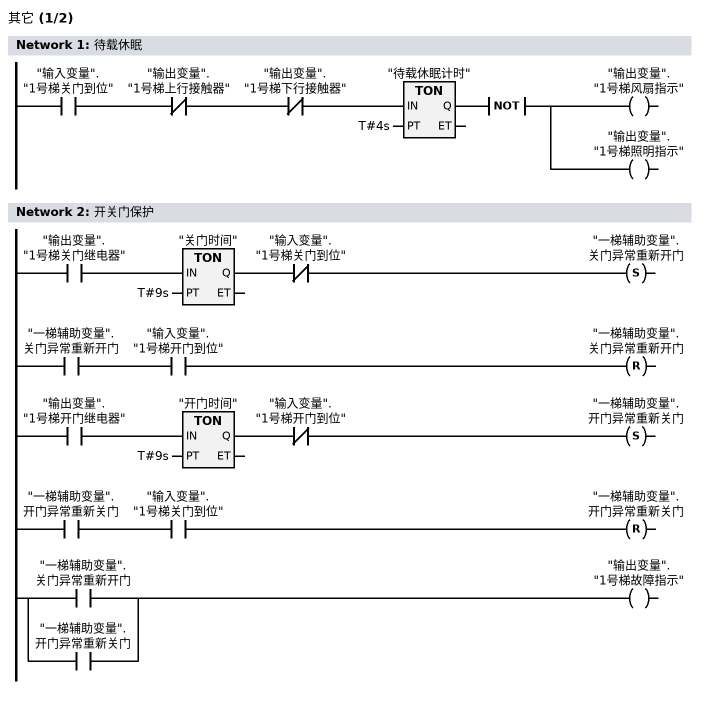
   "待载休眠计时".TON(IN := "输入变量"."1号梯关门到位" AND NOT "输出变量"."1号梯上行接触器" AND NOT "输出变量"."1号梯下行接触器", PT := T#4s);
   "输出变量"."1号梯风扇指示" := NOT "待载休眠计时".Q;
   "输出变量"."1号梯照明指示" := NOT "待载休眠计时".Q;
END_REGION

REGION Network 2: 开关门保护
   "关门时间".TON(IN := "输出变量"."1号梯关门继电器", PT := T#9s);
   IF "关门时间".Q AND NOT "输入变量"."1号梯关门到位" THEN "一梯辅助变量".关门异常重新开门 := TRUE; END_IF;
   IF "一梯辅助变量".关门异常重新开门 AND "输入变量"."1号梯开门到位" THEN "一梯辅助变量".关门异常重新开门 := FALSE; END_IF;
   "开门时间".TON(IN := "输出变量"."1号梯开门继电器", PT := T#9s);
   IF "开门时间".Q AND NOT "输入变量"."1号梯开门到位" THEN "一梯辅助变量".开门异常重新关门 := TRUE; END_IF;
   IF "一梯辅助变量".开门异常重新关门 AND "输入变量"."1号梯关门到位" THEN "一梯辅助变量".开门异常重新关门 := FALSE; END_IF;
   "输出变量"."1号梯故障指示" := "一梯辅助变量".关门异常重新开门 OR "一梯辅助变量".开门异常重新关门;
END_REGION

REGION Network 3: 限位保护
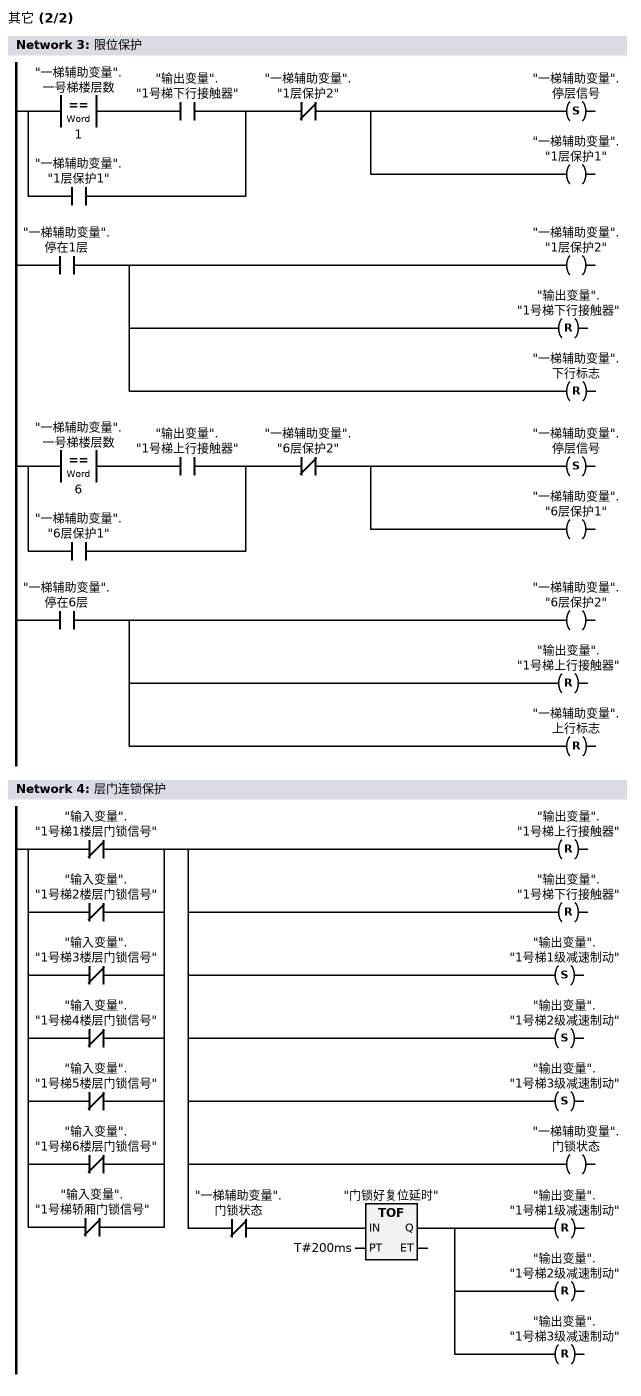
   RUNG wire#powerrail
      { S7_Templates := "SrcType := Word" } EQ_Contact(in1 := "一梯辅助变量".一号梯楼层数, in2 := 1)
      Contact( "输出变量"."1号梯下行接触器" )
      wire#w1
      I_Contact( "一梯辅助变量"."1层保护2" )
      wire#w2
      S_Coil( "一梯辅助变量".停层信号 )
   END_RUNG
   RUNG wire#powerrail
      Contact( "一梯辅助变量"."1层保护1" )
   END_RUNG wire#w1
   RUNG wire#w2
      Coil( "一梯辅助变量"."1层保护1" )
   END_RUNG
   RUNG wire#powerrail
      Contact( "一梯辅助变量".停在1层 )
      wire#w3
      Coil( "一梯辅助变量"."1层保护2" )
   END_RUNG
   RUNG wire#w3
      R_Coil( "输出变量"."1号梯下行接触器" )
   END_RUNG
   RUNG wire#w3
      R_Coil( "一梯辅助变量".下行标志 )
   END_RUNG
   RUNG wire#powerrail
      { S7_Templates := "SrcType := Word" } EQ_Contact(in1 := "一梯辅助变量".一号梯楼层数, in2 := 6)
      Contact( "输出变量"."1号梯上行接触器" )
      wire#w4
      I_Contact( "一梯辅助变量"."6层保护2" )
      wire#w5
      S_Coil( "一梯辅助变量".停层信号 )
   END_RUNG
   RUNG wire#powerrail
      Contact( "一梯辅助变量"."6层保护1" )
   END_RUNG wire#w4
   RUNG wire#w5
      Coil( "一梯辅助变量"."6层保护1" )
   END_RUNG
   RUNG wire#powerrail
      Contact( "一梯辅助变量".停在6层 )
      wire#w6
      Coil( "一梯辅助变量"."6层保护2" )
   END_RUNG
   RUNG wire#w6
      R_Coil( "输出变量"."1号梯上行接触器" )
   END_RUNG
   RUNG wire#w6
      R_Coil( "一梯辅助变量".上行标志 )
   END_RUNG
   // the same network as SCL:
   #_w1 := ((("一梯辅助变量".一号梯楼层数 = 1) AND "输出变量"."1号梯下行接触器") OR "一梯辅助变量"."1层保护1") AND NOT "一梯辅助变量"."1层保护2";
   IF #_w1 THEN "一梯辅助变量".停层信号 := TRUE; END_IF;
   "一梯辅助变量"."1层保护1" := #_w1;
   "一梯辅助变量"."1层保护2" := "一梯辅助变量".停在1层;
   IF "一梯辅助变量".停在1层 THEN
       "输出变量"."1号梯下行接触器" := FALSE;
       "一梯辅助变量".下行标志 := FALSE;
   END_IF;
   #_w2 := ((("一梯辅助变量".一号梯楼层数 = 6) AND "输出变量"."1号梯上行接触器") OR "一梯辅助变量"."6层保护1") AND NOT "一梯辅助变量"."6层保护2";
   IF #_w2 THEN "一梯辅助变量".停层信号 := TRUE; END_IF;
   "一梯辅助变量"."6层保护1" := #_w2;
   "一梯辅助变量"."6层保护2" := "一梯辅助变量".停在6层;
   IF "一梯辅助变量".停在6层 THEN
       "输出变量"."1号梯上行接触器" := FALSE;
       "一梯辅助变量".上行标志 := FALSE;
   END_IF;
END_REGION

REGION Network 4: 层门连锁保护
   #_w1 := NOT "输入变量"."1号梯1楼层门锁信号" OR NOT "输入变量"."1号梯2楼层门锁信号" OR NOT "输入变量"."1号梯3楼层门锁信号" OR NOT "输入变量"."1号梯4楼层门锁信号" OR NOT "输入变量"."1号梯5楼层门锁信号" OR NOT "输入变量"."1号梯6楼层门锁信号" OR NOT "输入变量"."1号梯轿厢门锁信号";
   IF #_w1 THEN
       "输出变量"."1号梯上行接触器" := FALSE;
       "输出变量"."1号梯下行接触器" := FALSE;
       "输出变量"."1号梯1级减速制动" := TRUE;
       "输出变量"."1号梯2级减速制动" := TRUE;
       "输出变量"."1号梯3级减速制动" := TRUE;
   END_IF;
   "一梯辅助变量".门锁状态 := #_w1;
   "门锁好复位延时".TOF(IN := #_w1 AND NOT "一梯辅助变量".门锁状态, PT := T#200ms);
   IF "门锁好复位延时".Q THEN
       "输出变量"."1号梯1级减速制动" := FALSE;
       "输出变量"."1号梯2级减速制动" := FALSE;
       "输出变量"."1号梯3级减速制动" := FALSE;
   END_IF;
END_REGION
END_FUNCTION

FUNCTION "初始化上行" : Void   // FC5, LAD
{ S7_Optimized_Access := 'TRUE' }
VERSION : 0.1
   VAR_TEMP   // added for the SCL form of the ladder/FBD networks
      _w1 : Bool;
   END_VAR
BEGIN

REGION Network 1: 按下按钮为1上行初始化
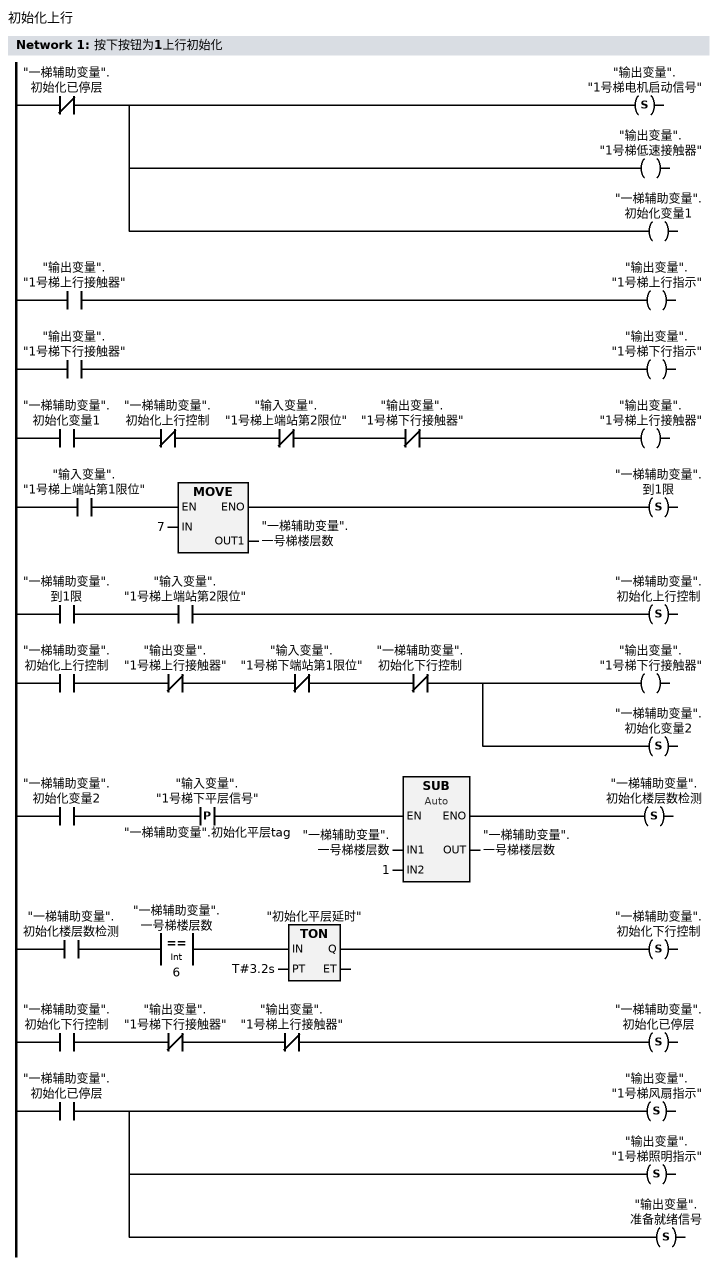
   IF NOT "一梯辅助变量".初始化已停层 THEN "输出变量"."1号梯电机启动信号" := TRUE; END_IF;
   "输出变量"."1号梯低速接触器" := NOT "一梯辅助变量".初始化已停层;
   "一梯辅助变量".初始化变量1 := NOT "一梯辅助变量".初始化已停层;
   "输出变量"."1号梯上行指示" := "输出变量"."1号梯上行接触器";
   "输出变量"."1号梯下行指示" := "输出变量"."1号梯下行接触器";
   "输出变量"."1号梯上行接触器" := "一梯辅助变量".初始化变量1 AND NOT "一梯辅助变量".初始化上行控制 AND NOT "输入变量"."1号梯上端站第2限位" AND NOT "输出变量"."1号梯下行接触器";
   IF "输入变量"."1号梯上端站第1限位" THEN
       "一梯辅助变量".一号梯楼层数 := 7;
       "一梯辅助变量".到1限 := TRUE;
   END_IF;
   IF "一梯辅助变量".到1限 AND "输入变量"."1号梯上端站第2限位" THEN "一梯辅助变量".初始化上行控制 := TRUE; END_IF;
   "输出变量"."1号梯下行接触器" := "一梯辅助变量".初始化上行控制 AND NOT "输出变量"."1号梯上行接触器" AND NOT "输入变量"."1号梯下端站第1限位" AND NOT "一梯辅助变量".初始化下行控制;
   IF "输出变量"."1号梯下行接触器" THEN "一梯辅助变量".初始化变量2 := TRUE; END_IF;
   #_w1 := "一梯辅助变量".初始化变量2 AND "输入变量"."1号梯下平层信号" AND NOT "一梯辅助变量".初始化平层tag;   // rising edge of "输入变量"."1号梯下平层信号"
   "一梯辅助变量".初始化平层tag := "输入变量"."1号梯下平层信号";
   IF #_w1 THEN
       "一梯辅助变量".一号梯楼层数 := "一梯辅助变量".一号梯楼层数 - 1;
       "一梯辅助变量".初始化楼层数检测 := TRUE;
   END_IF;
   "初始化平层延时".TON(IN := "一梯辅助变量".初始化楼层数检测 AND ("一梯辅助变量".一号梯楼层数 = 6), PT := T#3.2s);
   IF "初始化平层延时".Q THEN "一梯辅助变量".初始化下行控制 := TRUE; END_IF;
   IF "一梯辅助变量".初始化下行控制 AND NOT "输出变量"."1号梯下行接触器" AND NOT "输出变量"."1号梯上行接触器" THEN
       "一梯辅助变量".初始化已停层 := TRUE;
   END_IF;
   IF "一梯辅助变量".初始化已停层 THEN
       "输出变量"."1号梯风扇指示" := TRUE;
       "输出变量"."1号梯照明指示" := TRUE;
       "输出变量".准备就绪信号 := TRUE;
   END_IF;
END_REGION
END_FUNCTION

FUNCTION "上下行" : Void   // FC7, LAD
{ S7_Optimized_Access := 'TRUE' }
VERSION : 0.1
   VAR_TEMP   // added for the SCL form of the ladder/FBD networks
      _w1 : Bool;
      _w2 : Bool;
   END_VAR
BEGIN

REGION Network 1: 上行标志
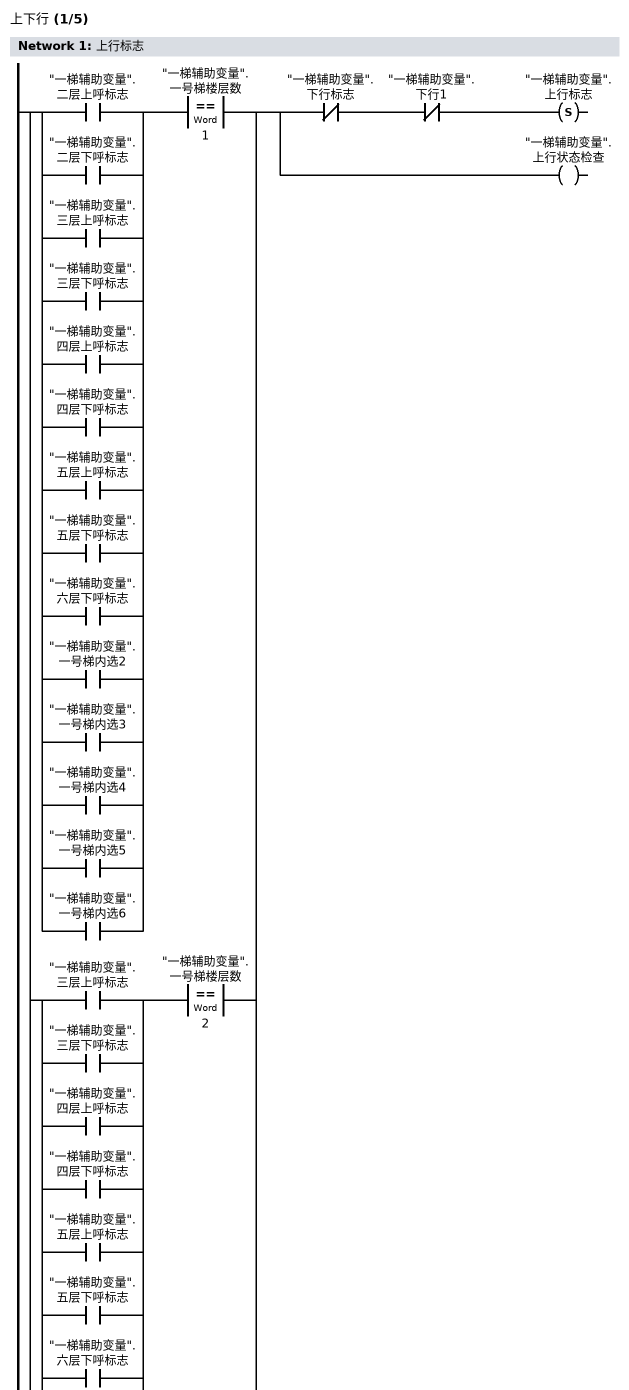
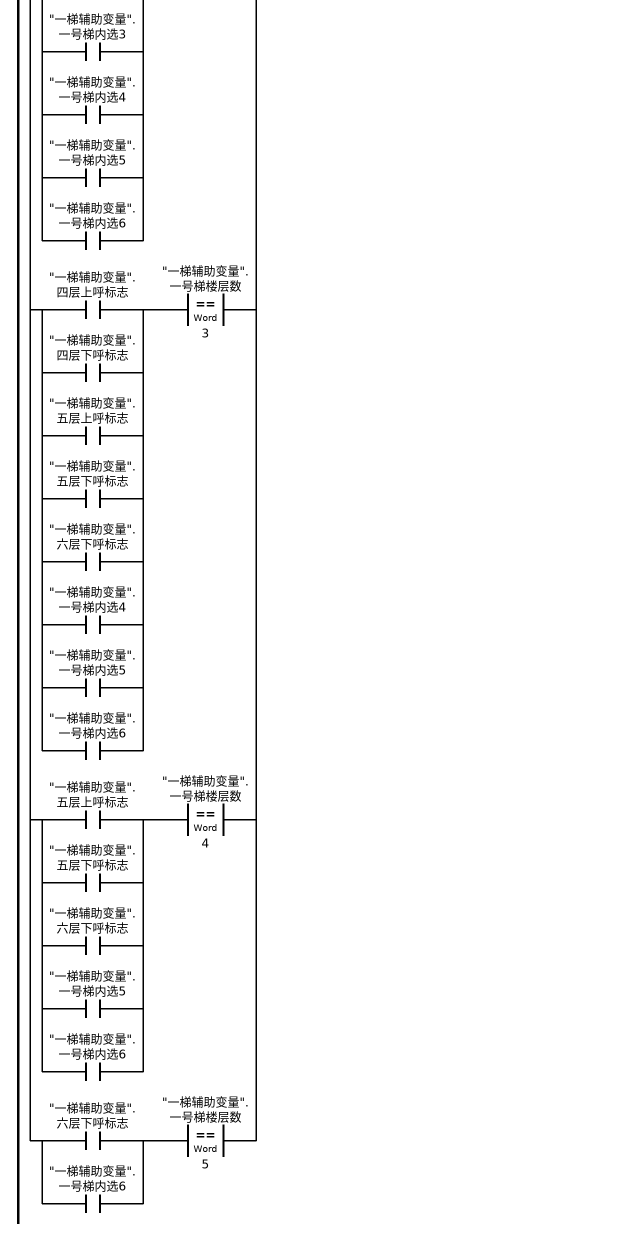
   RUNG wire#powerrail
      Contact( "一梯辅助变量".二层上呼标志 )
      wire#w1
      { S7_Templates := "SrcType := Word" } EQ_Contact(in1 := "一梯辅助变量".一号梯楼层数, in2 := 1)
      wire#w2
      I_Contact( "一梯辅助变量".下行标志 )
      I_Contact( "一梯辅助变量".下行1 )
      S_Coil( "一梯辅助变量".上行标志 )
   END_RUNG
   RUNG wire#powerrail
      Contact( "一梯辅助变量".二层下呼标志 )
   END_RUNG wire#w1
   RUNG wire#powerrail
      Contact( "一梯辅助变量".三层上呼标志 )
   END_RUNG wire#w1
   RUNG wire#powerrail
      Contact( "一梯辅助变量".三层下呼标志 )
   END_RUNG wire#w1
   RUNG wire#powerrail
      Contact( "一梯辅助变量".四层上呼标志 )
   END_RUNG wire#w1
   RUNG wire#powerrail
      Contact( "一梯辅助变量".四层下呼标志 )
   END_RUNG wire#w1
   RUNG wire#powerrail
      Contact( "一梯辅助变量".五层上呼标志 )
   END_RUNG wire#w1
   RUNG wire#powerrail
      Contact( "一梯辅助变量".五层下呼标志 )
   END_RUNG wire#w1
   RUNG wire#powerrail
      Contact( "一梯辅助变量".六层下呼标志 )
   END_RUNG wire#w1
   RUNG wire#powerrail
      Contact( "一梯辅助变量".一号梯内选2 )
   END_RUNG wire#w1
   RUNG wire#powerrail
      Contact( "一梯辅助变量".一号梯内选3 )
   END_RUNG wire#w1
   RUNG wire#powerrail
      Contact( "一梯辅助变量".一号梯内选4 )
   END_RUNG wire#w1
   RUNG wire#powerrail
      Contact( "一梯辅助变量".一号梯内选5 )
   END_RUNG wire#w1
   RUNG wire#powerrail
      Contact( "一梯辅助变量".一号梯内选6 )
   END_RUNG wire#w1
   RUNG wire#powerrail
      Contact( "一梯辅助变量".三层上呼标志 )
      wire#w3
      { S7_Templates := "SrcType := Word" } EQ_Contact(in1 := "一梯辅助变量".一号梯楼层数, in2 := 2)
   END_RUNG wire#w2
   RUNG wire#powerrail
      Contact( "一梯辅助变量".三层下呼标志 )
   END_RUNG wire#w3
   RUNG wire#powerrail
      Contact( "一梯辅助变量".四层上呼标志 )
   END_RUNG wire#w3
   RUNG wire#powerrail
      Contact( "一梯辅助变量".四层下呼标志 )
   END_RUNG wire#w3
   RUNG wire#powerrail
      Contact( "一梯辅助变量".五层上呼标志 )
   END_RUNG wire#w3
   RUNG wire#powerrail
      Contact( "一梯辅助变量".五层下呼标志 )
   END_RUNG wire#w3
   RUNG wire#powerrail
      Contact( "一梯辅助变量".六层下呼标志 )
   END_RUNG wire#w3
   RUNG wire#powerrail
      Contact( "一梯辅助变量".一号梯内选3 )
   END_RUNG wire#w3
   RUNG wire#powerrail
      Contact( "一梯辅助变量".一号梯内选4 )
   END_RUNG wire#w3
   RUNG wire#powerrail
      Contact( "一梯辅助变量".一号梯内选5 )
   END_RUNG wire#w3
   RUNG wire#powerrail
      Contact( "一梯辅助变量".一号梯内选6 )
   END_RUNG wire#w3
   RUNG wire#powerrail
      Contact( "一梯辅助变量".四层上呼标志 )
      wire#w4
      { S7_Templates := "SrcType := Word" } EQ_Contact(in1 := "一梯辅助变量".一号梯楼层数, in2 := 3)
   END_RUNG wire#w2
   RUNG wire#powerrail
      Contact( "一梯辅助变量".四层下呼标志 )
   END_RUNG wire#w4
   RUNG wire#powerrail
      Contact( "一梯辅助变量".五层上呼标志 )
   END_RUNG wire#w4
   RUNG wire#powerrail
      Contact( "一梯辅助变量".五层下呼标志 )
   END_RUNG wire#w4
   RUNG wire#powerrail
      Contact( "一梯辅助变量".六层下呼标志 )
   END_RUNG wire#w4
   RUNG wire#powerrail
      Contact( "一梯辅助变量".一号梯内选4 )
   END_RUNG wire#w4
   RUNG wire#powerrail
      Contact( "一梯辅助变量".一号梯内选5 )
   END_RUNG wire#w4
   RUNG wire#powerrail
      Contact( "一梯辅助变量".一号梯内选6 )
   END_RUNG wire#w4
   RUNG wire#powerrail
      Contact( "一梯辅助变量".五层上呼标志 )
      wire#w5
      { S7_Templates := "SrcType := Word" } EQ_Contact(in1 := "一梯辅助变量".一号梯楼层数, in2 := 4)
   END_RUNG wire#w2
   RUNG wire#powerrail
      Contact( "一梯辅助变量".五层下呼标志 )
   END_RUNG wire#w5
   RUNG wire#powerrail
      Contact( "一梯辅助变量".六层下呼标志 )
   END_RUNG wire#w5
   RUNG wire#powerrail
      Contact( "一梯辅助变量".一号梯内选5 )
   END_RUNG wire#w5
   RUNG wire#powerrail
      Contact( "一梯辅助变量".一号梯内选6 )
   END_RUNG wire#w5
   RUNG wire#powerrail
      Contact( "一梯辅助变量".六层下呼标志 )
      wire#w6
      { S7_Templates := "SrcType := Word" } EQ_Contact(in1 := "一梯辅助变量".一号梯楼层数, in2 := 5)
   END_RUNG wire#w2
   RUNG wire#powerrail
      Contact( "一梯辅助变量".一号梯内选6 )
   END_RUNG wire#w6
   RUNG wire#w2
      Coil( "一梯辅助变量".上行状态检查 )
   END_RUNG
   // the same network as SCL:
   #_w1 := (("一梯辅助变量".二层上呼标志 OR "一梯辅助变量".二层下呼标志 OR "一梯辅助变量".三层上呼标志 OR "一梯辅助变量".三层下呼标志 OR "一梯辅助变量".四层上呼标志 OR "一梯辅助变量".四层下呼标志 OR "一梯辅助变量".五层上呼标志 OR "一梯辅助变量".五层下呼标志 OR "一梯辅助变量".六层下呼标志 OR "一梯辅助变量".一号梯内选2 OR "一梯辅助变量".一号梯内选3 OR "一梯辅助变量".一号梯内选4 OR "一梯辅助变量".一号梯内选5 OR "一梯辅助变量".一号梯内选6) AND ("一梯辅助变量".一号梯楼层数 = 1)) OR (("一梯辅助变量".三层上呼标志 OR "一梯辅助变量".三层下呼标志 OR "一梯辅助变量".四层上呼标志 OR "一梯辅助变量".四层下呼标志 OR "一梯辅助变量".五层上呼标志 OR "一梯辅助变量".五层下呼标志 OR "一梯辅助变量".六层下呼标志 OR "一梯辅助变量".一号梯内选3 OR "一梯辅助变量".一号梯内选4 OR "一梯辅助变量".一号梯内选5 OR "一梯辅助变量".一号梯内选6) AND ("一梯辅助变量".一号梯楼层数 = 2)) OR (("一梯辅助变量".四层上呼标志 OR "一梯辅助变量".四层下呼标志 OR "一梯辅助变量".五层上呼标志 OR "一梯辅助变量".五层下呼标志 OR "一梯辅助变量".六层下呼标志 OR "一梯辅助变量".一号梯内选4 OR "一梯辅助变量".一号梯内选5 OR "一梯辅助变量".一号梯内选6) AND ("一梯辅助变量".一号梯楼层数 = 3)) OR (("一梯辅助变量".五层上呼标志 OR "一梯辅助变量".五层下呼标志 OR "一梯辅助变量".六层下呼标志 OR "一梯辅助变量".一号梯内选5 OR "一梯辅助变量".一号梯内选6) AND ("一梯辅助变量".一号梯楼层数 = 4)) OR (("一梯辅助变量".六层下呼标志 OR "一梯辅助变量".一号梯内选6) AND ("一梯辅助变量".一号梯楼层数 = 5));
   IF #_w1 AND NOT "一梯辅助变量".下行标志 AND NOT "一梯辅助变量".下行1 THEN "一梯辅助变量".上行标志 := TRUE; END_IF;
   "一梯辅助变量".上行状态检查 := #_w1;
END_REGION

REGION Network 2: 下行标志
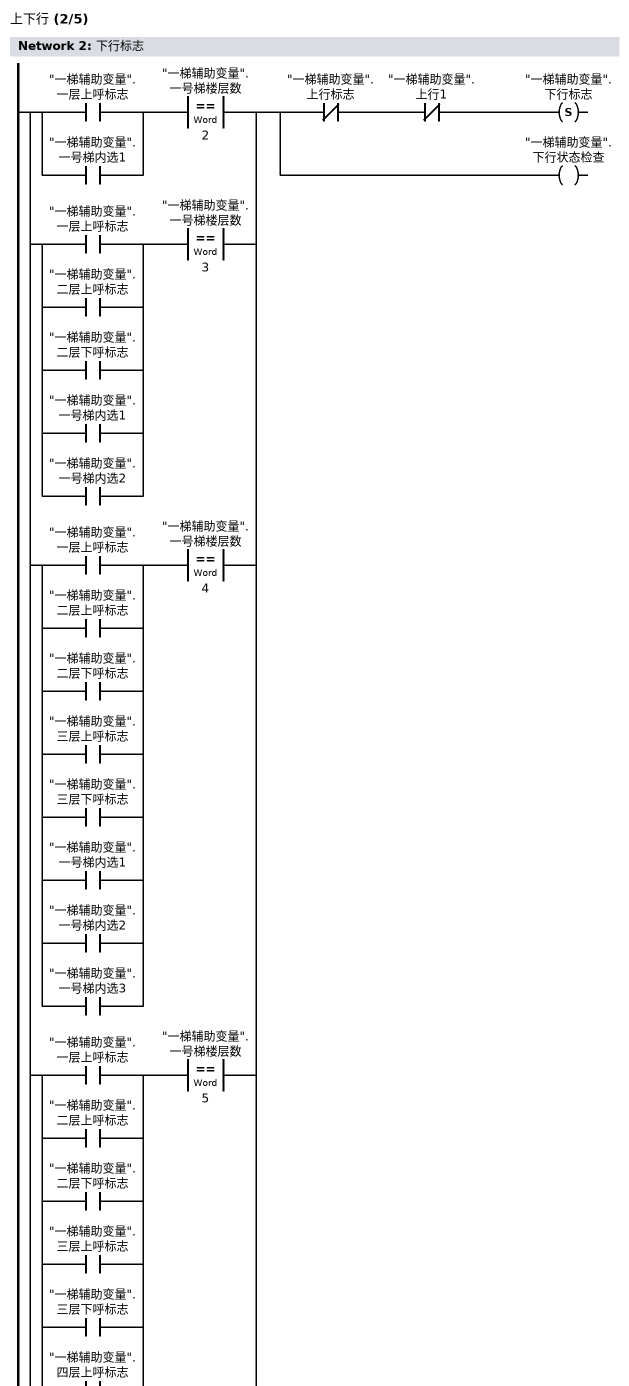
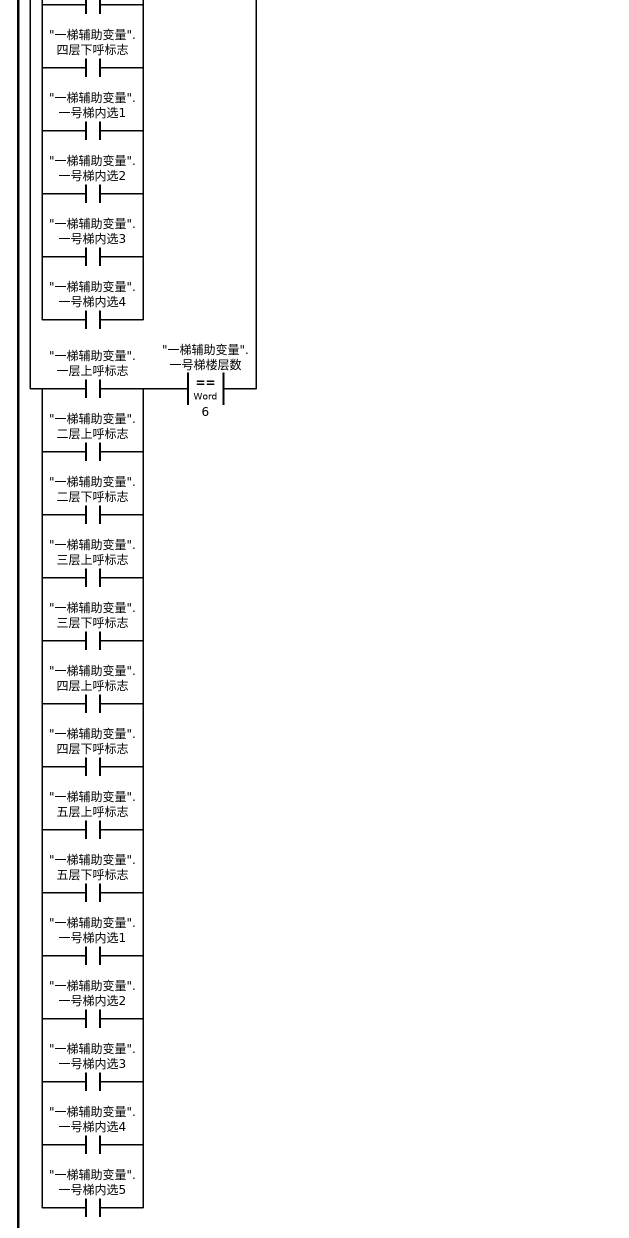
   RUNG wire#powerrail
      Contact( "一梯辅助变量".一层上呼标志 )
      wire#w1
      { S7_Templates := "SrcType := Word" } EQ_Contact(in1 := "一梯辅助变量".一号梯楼层数, in2 := 2)
      wire#w2
      I_Contact( "一梯辅助变量".上行标志 )
      I_Contact( "一梯辅助变量".上行1 )
      S_Coil( "一梯辅助变量".下行标志 )
   END_RUNG
   RUNG wire#powerrail
      Contact( "一梯辅助变量".一号梯内选1 )
   END_RUNG wire#w1
   RUNG wire#powerrail
      Contact( "一梯辅助变量".一层上呼标志 )
      wire#w3
      { S7_Templates := "SrcType := Word" } EQ_Contact(in1 := "一梯辅助变量".一号梯楼层数, in2 := 3)
   END_RUNG wire#w2
   RUNG wire#powerrail
      Contact( "一梯辅助变量".二层上呼标志 )
   END_RUNG wire#w3
   RUNG wire#powerrail
      Contact( "一梯辅助变量".二层下呼标志 )
   END_RUNG wire#w3
   RUNG wire#powerrail
      Contact( "一梯辅助变量".一号梯内选1 )
   END_RUNG wire#w3
   RUNG wire#powerrail
      Contact( "一梯辅助变量".一号梯内选2 )
   END_RUNG wire#w3
   RUNG wire#powerrail
      Contact( "一梯辅助变量".一层上呼标志 )
      wire#w4
      { S7_Templates := "SrcType := Word" } EQ_Contact(in1 := "一梯辅助变量".一号梯楼层数, in2 := 4)
   END_RUNG wire#w2
   RUNG wire#powerrail
      Contact( "一梯辅助变量".二层上呼标志 )
   END_RUNG wire#w4
   RUNG wire#powerrail
      Contact( "一梯辅助变量".二层下呼标志 )
   END_RUNG wire#w4
   RUNG wire#powerrail
      Contact( "一梯辅助变量".三层上呼标志 )
   END_RUNG wire#w4
   RUNG wire#powerrail
      Contact( "一梯辅助变量".三层下呼标志 )
   END_RUNG wire#w4
   RUNG wire#powerrail
      Contact( "一梯辅助变量".一号梯内选1 )
   END_RUNG wire#w4
   RUNG wire#powerrail
      Contact( "一梯辅助变量".一号梯内选2 )
   END_RUNG wire#w4
   RUNG wire#powerrail
      Contact( "一梯辅助变量".一号梯内选3 )
   END_RUNG wire#w4
   RUNG wire#powerrail
      Contact( "一梯辅助变量".一层上呼标志 )
      wire#w5
      { S7_Templates := "SrcType := Word" } EQ_Contact(in1 := "一梯辅助变量".一号梯楼层数, in2 := 5)
   END_RUNG wire#w2
   RUNG wire#powerrail
      Contact( "一梯辅助变量".二层上呼标志 )
   END_RUNG wire#w5
   RUNG wire#powerrail
      Contact( "一梯辅助变量".二层下呼标志 )
   END_RUNG wire#w5
   RUNG wire#powerrail
      Contact( "一梯辅助变量".三层上呼标志 )
   END_RUNG wire#w5
   RUNG wire#powerrail
      Contact( "一梯辅助变量".三层下呼标志 )
   END_RUNG wire#w5
   RUNG wire#powerrail
      Contact( "一梯辅助变量".四层上呼标志 )
   END_RUNG wire#w5
   RUNG wire#powerrail
      Contact( "一梯辅助变量".四层下呼标志 )
   END_RUNG wire#w5
   RUNG wire#powerrail
      Contact( "一梯辅助变量".一号梯内选1 )
   END_RUNG wire#w5
   RUNG wire#powerrail
      Contact( "一梯辅助变量".一号梯内选2 )
   END_RUNG wire#w5
   RUNG wire#powerrail
      Contact( "一梯辅助变量".一号梯内选3 )
   END_RUNG wire#w5
   RUNG wire#powerrail
      Contact( "一梯辅助变量".一号梯内选4 )
   END_RUNG wire#w5
   RUNG wire#powerrail
      Contact( "一梯辅助变量".一层上呼标志 )
      wire#w6
      { S7_Templates := "SrcType := Word" } EQ_Contact(in1 := "一梯辅助变量".一号梯楼层数, in2 := 6)
   END_RUNG wire#w2
   RUNG wire#powerrail
      Contact( "一梯辅助变量".二层上呼标志 )
   END_RUNG wire#w6
   RUNG wire#powerrail
      Contact( "一梯辅助变量".二层下呼标志 )
   END_RUNG wire#w6
   RUNG wire#powerrail
      Contact( "一梯辅助变量".三层上呼标志 )
   END_RUNG wire#w6
   RUNG wire#powerrail
      Contact( "一梯辅助变量".三层下呼标志 )
   END_RUNG wire#w6
   RUNG wire#powerrail
      Contact( "一梯辅助变量".四层上呼标志 )
   END_RUNG wire#w6
   RUNG wire#powerrail
      Contact( "一梯辅助变量".四层下呼标志 )
   END_RUNG wire#w6
   RUNG wire#powerrail
      Contact( "一梯辅助变量".五层上呼标志 )
   END_RUNG wire#w6
   RUNG wire#powerrail
      Contact( "一梯辅助变量".五层下呼标志 )
   END_RUNG wire#w6
   RUNG wire#powerrail
      Contact( "一梯辅助变量".一号梯内选1 )
   END_RUNG wire#w6
   RUNG wire#powerrail
      Contact( "一梯辅助变量".一号梯内选2 )
   END_RUNG wire#w6
   RUNG wire#powerrail
      Contact( "一梯辅助变量".一号梯内选3 )
   END_RUNG wire#w6
   RUNG wire#powerrail
      Contact( "一梯辅助变量".一号梯内选4 )
   END_RUNG wire#w6
   RUNG wire#powerrail
      Contact( "一梯辅助变量".一号梯内选5 )
   END_RUNG wire#w6
   RUNG wire#w2
      Coil( "一梯辅助变量".下行状态检查 )
   END_RUNG
   // the same network as SCL:
   #_w1 := (("一梯辅助变量".一层上呼标志 OR "一梯辅助变量".一号梯内选1) AND ("一梯辅助变量".一号梯楼层数 = 2)) OR (("一梯辅助变量".一层上呼标志 OR "一梯辅助变量".二层上呼标志 OR "一梯辅助变量".二层下呼标志 OR "一梯辅助变量".一号梯内选1 OR "一梯辅助变量".一号梯内选2) AND ("一梯辅助变量".一号梯楼层数 = 3)) OR (("一梯辅助变量".一层上呼标志 OR "一梯辅助变量".二层上呼标志 OR "一梯辅助变量".二层下呼标志 OR "一梯辅助变量".三层上呼标志 OR "一梯辅助变量".三层下呼标志 OR "一梯辅助变量".一号梯内选1 OR "一梯辅助变量".一号梯内选2 OR "一梯辅助变量".一号梯内选3) AND ("一梯辅助变量".一号梯楼层数 = 4)) OR (("一梯辅助变量".一层上呼标志 OR "一梯辅助变量".二层上呼标志 OR "一梯辅助变量".二层下呼标志 OR "一梯辅助变量".三层上呼标志 OR "一梯辅助变量".三层下呼标志 OR "一梯辅助变量".四层上呼标志 OR "一梯辅助变量".四层下呼标志 OR "一梯辅助变量".一号梯内选1 OR "一梯辅助变量".一号梯内选2 OR "一梯辅助变量".一号梯内选3 OR "一梯辅助变量".一号梯内选4) AND ("一梯辅助变量".一号梯楼层数 = 5)) OR (("一梯辅助变量".一层上呼标志 OR "一梯辅助变量".二层上呼标志 OR "一梯辅助变量".二层下呼标志 OR "一梯辅助变量".三层上呼标志 OR "一梯辅助变量".三层下呼标志 OR "一梯辅助变量".四层上呼标志 OR "一梯辅助变量".四层下呼标志 OR "一梯辅助变量".五层上呼标志 OR "一梯辅助变量".五层下呼标志 OR "一梯辅助变量".一号梯内选1 OR "一梯辅助变量".一号梯内选2 OR "一梯辅助变量".一号梯内选3 OR "一梯辅助变量".一号梯内选4 OR "一梯辅助变量".一号梯内选5) AND ("一梯辅助变量".一号梯楼层数 = 6));
   IF #_w1 AND NOT "一梯辅助变量".上行标志 AND NOT "一梯辅助变量".上行1 THEN "一梯辅助变量".下行标志 := TRUE; END_IF;
   "一梯辅助变量".下行状态检查 := #_w1;
END_REGION

REGION Network 3: 楼层计数
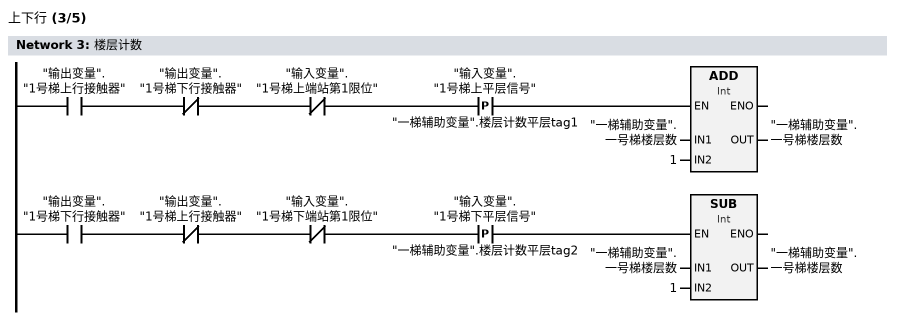
   RUNG wire#powerrail
      Contact( "输出变量"."1号梯上行接触器" )
      I_Contact( "输出变量"."1号梯下行接触器" )
      I_Contact( "输入变量"."1号梯上端站第1限位" )
      P_Contact(operand := "输入变量"."1号梯上平层信号", bit := "一梯辅助变量".楼层计数平层tag1)
      { S7_Templates := "SrcType := Int" } Add(in1 := "一梯辅助变量".一号梯楼层数, in2 := 1, out => "一梯辅助变量".一号梯楼层数)
   END_RUNG
   RUNG wire#powerrail
      Contact( "输出变量"."1号梯下行接触器" )
      I_Contact( "输出变量"."1号梯上行接触器" )
      I_Contact( "输入变量"."1号梯下端站第1限位" )
      P_Contact(operand := "输入变量"."1号梯下平层信号", bit := "一梯辅助变量".楼层计数平层tag2)
      { S7_Templates := "SrcType := Int" } Sub(in1 := "一梯辅助变量".一号梯楼层数, in2 := 1, out => "一梯辅助变量".一号梯楼层数)
   END_RUNG
   // the same network as SCL:
   #_w1 := "输出变量"."1号梯上行接触器" AND NOT "输出变量"."1号梯下行接触器" AND NOT "输入变量"."1号梯上端站第1限位" AND "输入变量"."1号梯上平层信号" AND NOT "一梯辅助变量".楼层计数平层tag1;   // rising edge of "输入变量"."1号梯上平层信号"
   "一梯辅助变量".楼层计数平层tag1 := "输入变量"."1号梯上平层信号";
   IF #_w1 THEN "一梯辅助变量".一号梯楼层数 := "一梯辅助变量".一号梯楼层数 + 1; END_IF;
   #_w2 := "输出变量"."1号梯下行接触器" AND NOT "输出变量"."1号梯上行接触器" AND NOT "输入变量"."1号梯下端站第1限位" AND "输入变量"."1号梯下平层信号" AND NOT "一梯辅助变量".楼层计数平层tag2;   // rising edge of "输入变量"."1号梯下平层信号"
   "一梯辅助变量".楼层计数平层tag2 := "输入变量"."1号梯下平层信号";
   IF #_w2 THEN "一梯辅助变量".一号梯楼层数 := "一梯辅助变量".一号梯楼层数 - 1; END_IF;
END_REGION

REGION Network 4: 上下行标志及灯
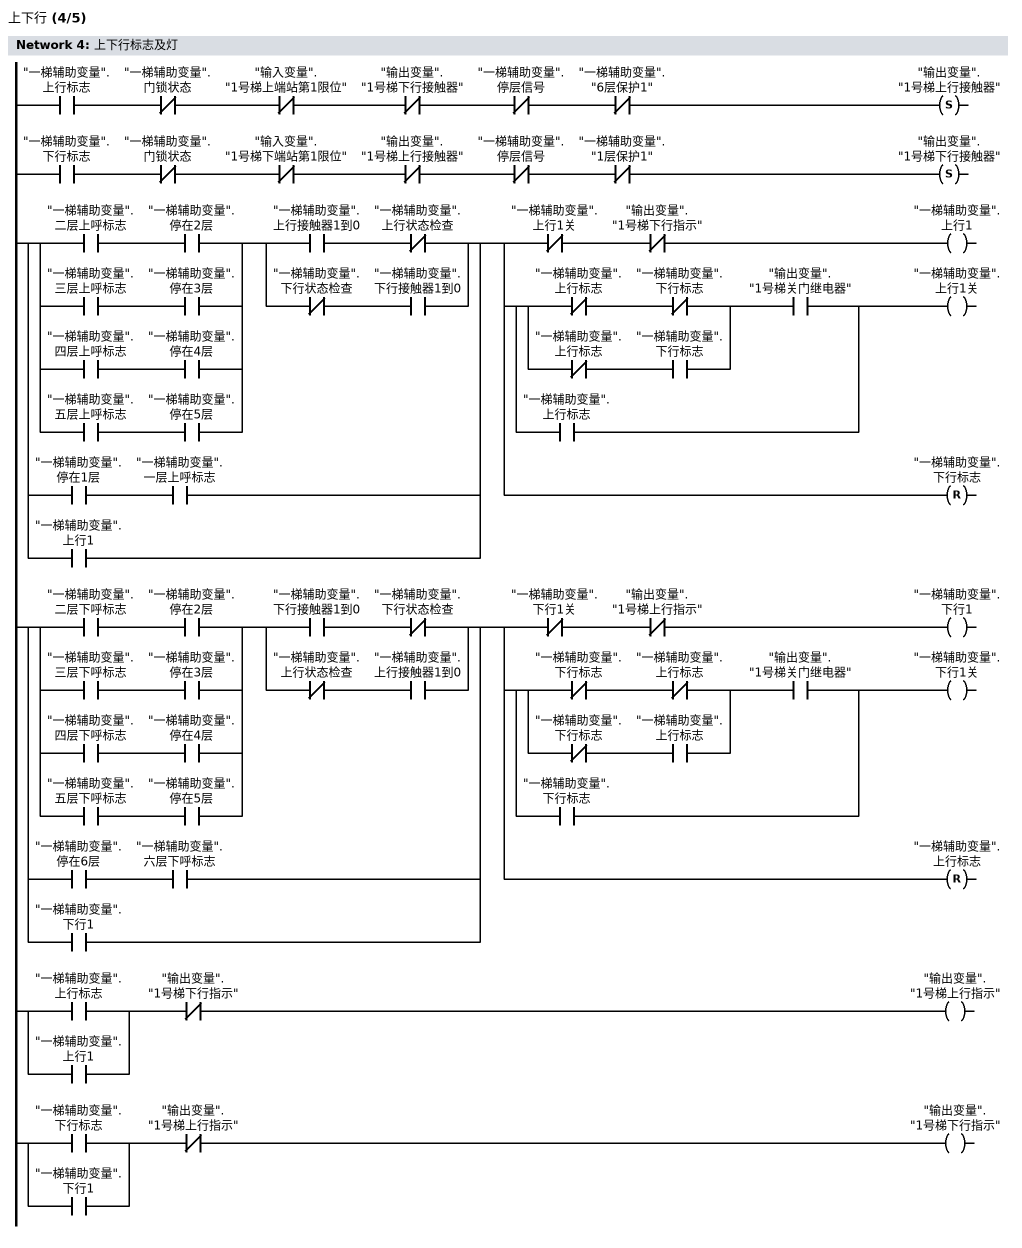
   RUNG wire#powerrail
      Contact( "一梯辅助变量".上行标志 )
      I_Contact( "一梯辅助变量".门锁状态 )
      I_Contact( "输入变量"."1号梯上端站第1限位" )
      I_Contact( "输出变量"."1号梯下行接触器" )
      I_Contact( "一梯辅助变量".停层信号 )
      I_Contact( "一梯辅助变量"."6层保护1" )
      S_Coil( "输出变量"."1号梯上行接触器" )
   END_RUNG
   RUNG wire#powerrail
      Contact( "一梯辅助变量".下行标志 )
      I_Contact( "一梯辅助变量".门锁状态 )
      I_Contact( "输入变量"."1号梯下端站第1限位" )
      I_Contact( "输出变量"."1号梯上行接触器" )
      I_Contact( "一梯辅助变量".停层信号 )
      I_Contact( "一梯辅助变量"."1层保护1" )
      S_Coil( "输出变量"."1号梯下行接触器" )
   END_RUNG
   RUNG wire#powerrail
      Contact( "一梯辅助变量".二层上呼标志 )
      Contact( "一梯辅助变量".停在2层 )
      wire#w1
      Contact( "一梯辅助变量".上行接触器1到0 )
      I_Contact( "一梯辅助变量".上行状态检查 )
      wire#w2
      I_Contact( "一梯辅助变量".上行1关 )
      I_Contact( "输出变量"."1号梯下行指示" )
      Coil( "一梯辅助变量".上行1 )
   END_RUNG
   RUNG wire#powerrail
      Contact( "一梯辅助变量".三层上呼标志 )
      Contact( "一梯辅助变量".停在3层 )
   END_RUNG wire#w1
   RUNG wire#powerrail
      Contact( "一梯辅助变量".四层上呼标志 )
      Contact( "一梯辅助变量".停在4层 )
   END_RUNG wire#w1
   RUNG wire#powerrail
      Contact( "一梯辅助变量".五层上呼标志 )
      Contact( "一梯辅助变量".停在5层 )
   END_RUNG wire#w1
   RUNG wire#w1
      I_Contact( "一梯辅助变量".下行状态检查 )
      Contact( "一梯辅助变量".下行接触器1到0 )
   END_RUNG wire#w2
   RUNG wire#powerrail
      Contact( "一梯辅助变量".停在1层 )
      Contact( "一梯辅助变量".一层上呼标志 )
   END_RUNG wire#w2
   RUNG wire#powerrail
      Contact( "一梯辅助变量".上行1 )
   END_RUNG wire#w2
   RUNG wire#w2
      I_Contact( "一梯辅助变量".上行标志 )
      I_Contact( "一梯辅助变量".下行标志 )
      wire#w3
      Contact( "输出变量"."1号梯关门继电器" )
      wire#w4
      Coil( "一梯辅助变量".上行1关 )
   END_RUNG
   RUNG wire#w2
      I_Contact( "一梯辅助变量".上行标志 )
      Contact( "一梯辅助变量".下行标志 )
   END_RUNG wire#w3
   RUNG wire#w2
      Contact( "一梯辅助变量".上行标志 )
   END_RUNG wire#w4
   RUNG wire#w2
      R_Coil( "一梯辅助变量".下行标志 )
   END_RUNG
   RUNG wire#powerrail
      Contact( "一梯辅助变量".二层下呼标志 )
      Contact( "一梯辅助变量".停在2层 )
      wire#w5
      Contact( "一梯辅助变量".下行接触器1到0 )
      I_Contact( "一梯辅助变量".下行状态检查 )
      wire#w6
      I_Contact( "一梯辅助变量".下行1关 )
      I_Contact( "输出变量"."1号梯上行指示" )
      Coil( "一梯辅助变量".下行1 )
   END_RUNG
   RUNG wire#powerrail
      Contact( "一梯辅助变量".三层下呼标志 )
      Contact( "一梯辅助变量".停在3层 )
   END_RUNG wire#w5
   RUNG wire#powerrail
      Contact( "一梯辅助变量".四层下呼标志 )
      Contact( "一梯辅助变量".停在4层 )
   END_RUNG wire#w5
   RUNG wire#powerrail
      Contact( "一梯辅助变量".五层下呼标志 )
      Contact( "一梯辅助变量".停在5层 )
   END_RUNG wire#w5
   RUNG wire#w5
      I_Contact( "一梯辅助变量".上行状态检查 )
      Contact( "一梯辅助变量".上行接触器1到0 )
   END_RUNG wire#w6
   RUNG wire#powerrail
      Contact( "一梯辅助变量".停在6层 )
      Contact( "一梯辅助变量".六层下呼标志 )
   END_RUNG wire#w6
   RUNG wire#powerrail
      Contact( "一梯辅助变量".下行1 )
   END_RUNG wire#w6
   RUNG wire#w6
      I_Contact( "一梯辅助变量".下行标志 )
      I_Contact( "一梯辅助变量".上行标志 )
      wire#w7
      Contact( "输出变量"."1号梯关门继电器" )
      wire#w8
      Coil( "一梯辅助变量".下行1关 )
   END_RUNG
   RUNG wire#w6
      I_Contact( "一梯辅助变量".下行标志 )
      Contact( "一梯辅助变量".上行标志 )
   END_RUNG wire#w7
   RUNG wire#w6
      Contact( "一梯辅助变量".下行标志 )
   END_RUNG wire#w8
   RUNG wire#w6
      R_Coil( "一梯辅助变量".上行标志 )
   END_RUNG
   RUNG wire#powerrail
      Contact( "一梯辅助变量".上行标志 )
      wire#w9
      I_Contact( "输出变量"."1号梯下行指示" )
      Coil( "输出变量"."1号梯上行指示" )
   END_RUNG
   RUNG wire#powerrail
      Contact( "一梯辅助变量".上行1 )
   END_RUNG wire#w9
   RUNG wire#powerrail
      Contact( "一梯辅助变量".下行标志 )
      wire#w10
      I_Contact( "输出变量"."1号梯上行指示" )
      Coil( "输出变量"."1号梯下行指示" )
   END_RUNG
   RUNG wire#powerrail
      Contact( "一梯辅助变量".下行1 )
   END_RUNG wire#w10
   // the same network as SCL:
   IF "一梯辅助变量".上行标志 AND NOT "一梯辅助变量".门锁状态 AND NOT "输入变量"."1号梯上端站第1限位" AND NOT "输出变量"."1号梯下行接触器" AND NOT "一梯辅助变量".停层信号 AND NOT "一梯辅助变量"."6层保护1" THEN
       "输出变量"."1号梯上行接触器" := TRUE;
   END_IF;
   IF "一梯辅助变量".下行标志 AND NOT "一梯辅助变量".门锁状态 AND NOT "输入变量"."1号梯下端站第1限位" AND NOT "输出变量"."1号梯上行接触器" AND NOT "一梯辅助变量".停层信号 AND NOT "一梯辅助变量"."1层保护1" THEN
       "输出变量"."1号梯下行接触器" := TRUE;
   END_IF;
   #_w1 := ((("一梯辅助变量".二层上呼标志 AND "一梯辅助变量".停在2层) OR ("一梯辅助变量".三层上呼标志 AND "一梯辅助变量".停在3层) OR ("一梯辅助变量".四层上呼标志 AND "一梯辅助变量".停在4层) OR ("一梯辅助变量".五层上呼标志 AND "一梯辅助变量".停在5层)) AND (("一梯辅助变量".上行接触器1到0 AND NOT "一梯辅助变量".上行状态检查) OR (NOT "一梯辅助变量".下行状态检查 AND "一梯辅助变量".下行接触器1到0))) OR ("一梯辅助变量".停在1层 AND "一梯辅助变量".一层上呼标志) OR "一梯辅助变量".上行1;
   "一梯辅助变量".上行1 := #_w1 AND NOT "一梯辅助变量".上行1关 AND NOT "输出变量"."1号梯下行指示";
   "一梯辅助变量".上行1关 := #_w1 AND ((((NOT "一梯辅助变量".上行标志 AND NOT "一梯辅助变量".下行标志) OR (NOT "一梯辅助变量".上行标志 AND "一梯辅助变量".下行标志)) AND "输出变量"."1号梯关门继电器") OR "一梯辅助变量".上行标志);
   IF #_w1 THEN "一梯辅助变量".下行标志 := FALSE; END_IF;
   #_w2 := ((("一梯辅助变量".二层下呼标志 AND "一梯辅助变量".停在2层) OR ("一梯辅助变量".三层下呼标志 AND "一梯辅助变量".停在3层) OR ("一梯辅助变量".四层下呼标志 AND "一梯辅助变量".停在4层) OR ("一梯辅助变量".五层下呼标志 AND "一梯辅助变量".停在5层)) AND (("一梯辅助变量".下行接触器1到0 AND NOT "一梯辅助变量".下行状态检查) OR (NOT "一梯辅助变量".上行状态检查 AND "一梯辅助变量".上行接触器1到0))) OR ("一梯辅助变量".停在6层 AND "一梯辅助变量".六层下呼标志) OR "一梯辅助变量".下行1;
   "一梯辅助变量".下行1 := #_w2 AND NOT "一梯辅助变量".下行1关 AND NOT "输出变量"."1号梯上行指示";
   "一梯辅助变量".下行1关 := #_w2 AND ((((NOT "一梯辅助变量".下行标志 AND NOT "一梯辅助变量".上行标志) OR (NOT "一梯辅助变量".下行标志 AND "一梯辅助变量".上行标志)) AND "输出变量"."1号梯关门继电器") OR "一梯辅助变量".下行标志);
   IF #_w2 THEN "一梯辅助变量".上行标志 := FALSE; END_IF;
   "输出变量"."1号梯上行指示" := ("一梯辅助变量".上行标志 OR "一梯辅助变量".上行1) AND NOT "输出变量"."1号梯下行指示";
   "输出变量"."1号梯下行指示" := ("一梯辅助变量".下行标志 OR "一梯辅助变量".下行1) AND NOT "输出变量"."1号梯上行指示";
END_REGION

REGION Network 5: 数码管显示楼层
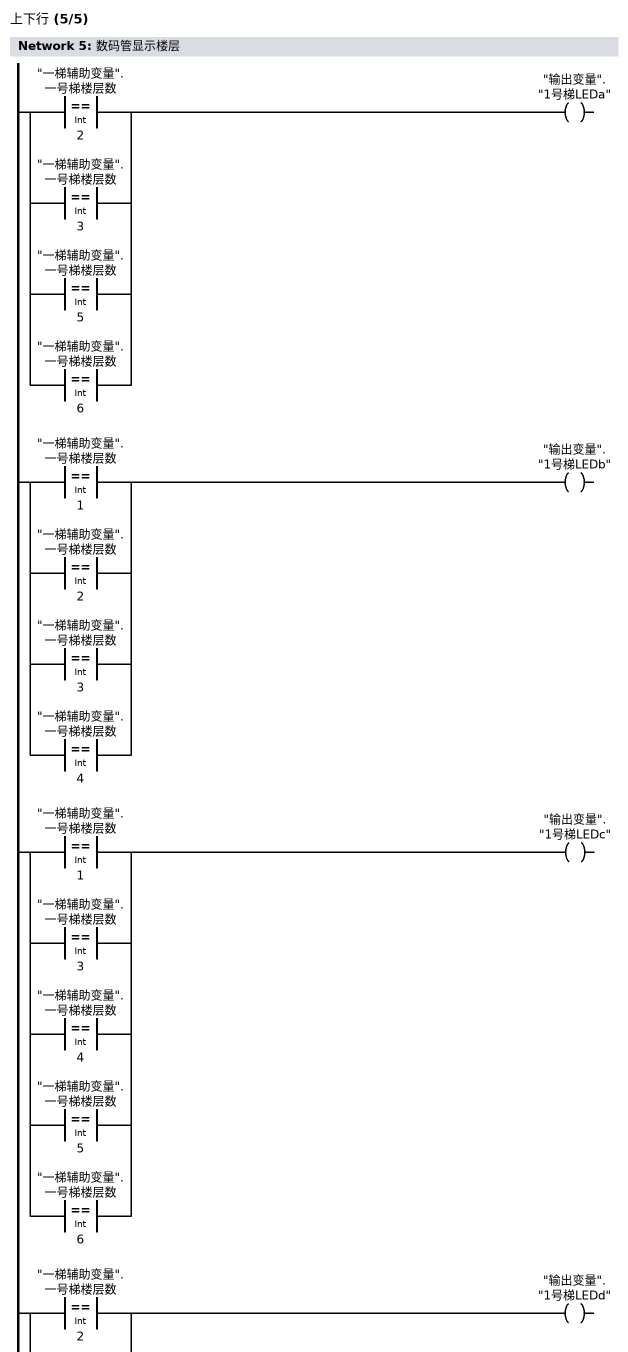
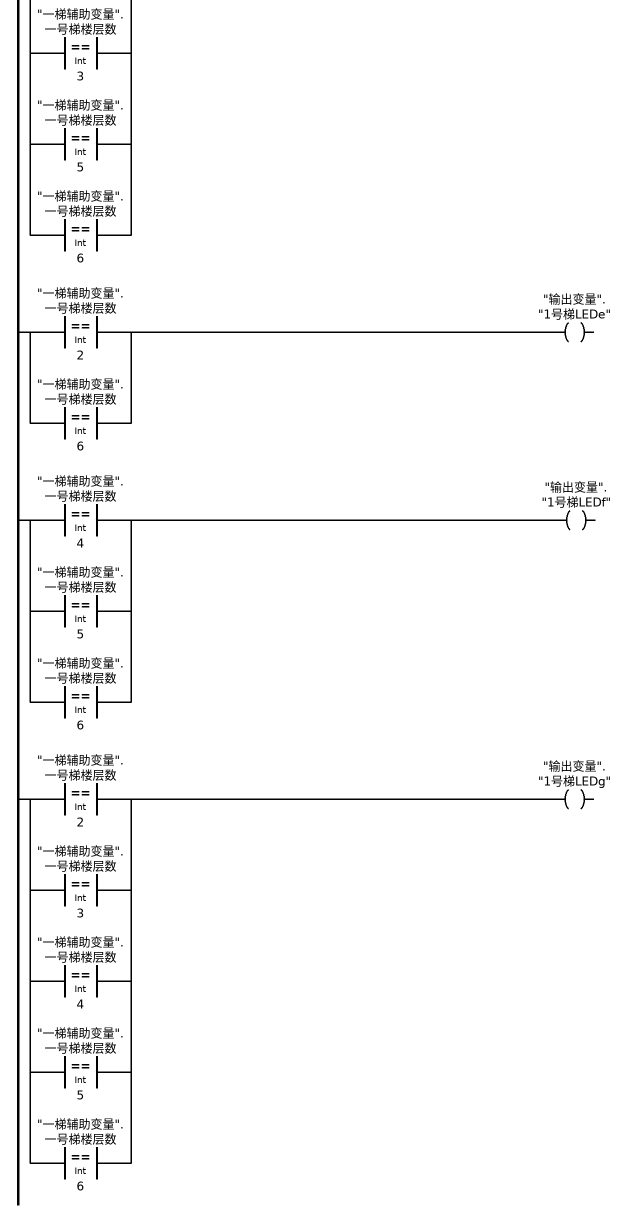
   RUNG wire#powerrail
      { S7_Templates := "SrcType := Int" } EQ_Contact(in1 := "一梯辅助变量".一号梯楼层数, in2 := 2)
      wire#w1
      Coil( "输出变量"."1号梯LEDa" )
   END_RUNG
   RUNG wire#powerrail
      { S7_Templates := "SrcType := Int" } EQ_Contact(in1 := "一梯辅助变量".一号梯楼层数, in2 := 3)
   END_RUNG wire#w1
   RUNG wire#powerrail
      { S7_Templates := "SrcType := Int" } EQ_Contact(in1 := "一梯辅助变量".一号梯楼层数, in2 := 5)
   END_RUNG wire#w1
   RUNG wire#powerrail
      { S7_Templates := "SrcType := Int" } EQ_Contact(in1 := "一梯辅助变量".一号梯楼层数, in2 := 6)
   END_RUNG wire#w1
   RUNG wire#powerrail
      { S7_Templates := "SrcType := Int" } EQ_Contact(in1 := "一梯辅助变量".一号梯楼层数, in2 := 1)
      wire#w2
      Coil( "输出变量"."1号梯LEDb" )
   END_RUNG
   RUNG wire#powerrail
      { S7_Templates := "SrcType := Int" } EQ_Contact(in1 := "一梯辅助变量".一号梯楼层数, in2 := 2)
   END_RUNG wire#w2
   RUNG wire#powerrail
      { S7_Templates := "SrcType := Int" } EQ_Contact(in1 := "一梯辅助变量".一号梯楼层数, in2 := 3)
   END_RUNG wire#w2
   RUNG wire#powerrail
      { S7_Templates := "SrcType := Int" } EQ_Contact(in1 := "一梯辅助变量".一号梯楼层数, in2 := 4)
   END_RUNG wire#w2
   RUNG wire#powerrail
      { S7_Templates := "SrcType := Int" } EQ_Contact(in1 := "一梯辅助变量".一号梯楼层数, in2 := 1)
      wire#w3
      Coil( "输出变量"."1号梯LEDc" )
   END_RUNG
   RUNG wire#powerrail
      { S7_Templates := "SrcType := Int" } EQ_Contact(in1 := "一梯辅助变量".一号梯楼层数, in2 := 3)
   END_RUNG wire#w3
   RUNG wire#powerrail
      { S7_Templates := "SrcType := Int" } EQ_Contact(in1 := "一梯辅助变量".一号梯楼层数, in2 := 4)
   END_RUNG wire#w3
   RUNG wire#powerrail
      { S7_Templates := "SrcType := Int" } EQ_Contact(in1 := "一梯辅助变量".一号梯楼层数, in2 := 5)
   END_RUNG wire#w3
   RUNG wire#powerrail
      { S7_Templates := "SrcType := Int" } EQ_Contact(in1 := "一梯辅助变量".一号梯楼层数, in2 := 6)
   END_RUNG wire#w3
   RUNG wire#powerrail
      { S7_Templates := "SrcType := Int" } EQ_Contact(in1 := "一梯辅助变量".一号梯楼层数, in2 := 2)
      wire#w4
      Coil( "输出变量"."1号梯LEDd" )
   END_RUNG
   RUNG wire#powerrail
      { S7_Templates := "SrcType := Int" } EQ_Contact(in1 := "一梯辅助变量".一号梯楼层数, in2 := 3)
   END_RUNG wire#w4
   RUNG wire#powerrail
      { S7_Templates := "SrcType := Int" } EQ_Contact(in1 := "一梯辅助变量".一号梯楼层数, in2 := 5)
   END_RUNG wire#w4
   RUNG wire#powerrail
      { S7_Templates := "SrcType := Int" } EQ_Contact(in1 := "一梯辅助变量".一号梯楼层数, in2 := 6)
   END_RUNG wire#w4
   RUNG wire#powerrail
      { S7_Templates := "SrcType := Int" } EQ_Contact(in1 := "一梯辅助变量".一号梯楼层数, in2 := 2)
      wire#w5
      Coil( "输出变量"."1号梯LEDe" )
   END_RUNG
   RUNG wire#powerrail
      { S7_Templates := "SrcType := Int" } EQ_Contact(in1 := "一梯辅助变量".一号梯楼层数, in2 := 6)
   END_RUNG wire#w5
   RUNG wire#powerrail
      { S7_Templates := "SrcType := Int" } EQ_Contact(in1 := "一梯辅助变量".一号梯楼层数, in2 := 4)
      wire#w6
      Coil( "输出变量"."1号梯LEDf" )
   END_RUNG
   RUNG wire#powerrail
      { S7_Templates := "SrcType := Int" } EQ_Contact(in1 := "一梯辅助变量".一号梯楼层数, in2 := 5)
   END_RUNG wire#w6
   RUNG wire#powerrail
      { S7_Templates := "SrcType := Int" } EQ_Contact(in1 := "一梯辅助变量".一号梯楼层数, in2 := 6)
   END_RUNG wire#w6
   RUNG wire#powerrail
      { S7_Templates := "SrcType := Int" } EQ_Contact(in1 := "一梯辅助变量".一号梯楼层数, in2 := 2)
      wire#w7
      Coil( "输出变量"."1号梯LEDg" )
   END_RUNG
   RUNG wire#powerrail
      { S7_Templates := "SrcType := Int" } EQ_Contact(in1 := "一梯辅助变量".一号梯楼层数, in2 := 3)
   END_RUNG wire#w7
   RUNG wire#powerrail
      { S7_Templates := "SrcType := Int" } EQ_Contact(in1 := "一梯辅助变量".一号梯楼层数, in2 := 4)
   END_RUNG wire#w7
   RUNG wire#powerrail
      { S7_Templates := "SrcType := Int" } EQ_Contact(in1 := "一梯辅助变量".一号梯楼层数, in2 := 5)
   END_RUNG wire#w7
   RUNG wire#powerrail
      { S7_Templates := "SrcType := Int" } EQ_Contact(in1 := "一梯辅助变量".一号梯楼层数, in2 := 6)
   END_RUNG wire#w7
   // the same network as SCL:
   "输出变量"."1号梯LEDa" := ("一梯辅助变量".一号梯楼层数 = 2) OR ("一梯辅助变量".一号梯楼层数 = 3) OR ("一梯辅助变量".一号梯楼层数 = 5) OR ("一梯辅助变量".一号梯楼层数 = 6);
   "输出变量"."1号梯LEDb" := ("一梯辅助变量".一号梯楼层数 = 1) OR ("一梯辅助变量".一号梯楼层数 = 2) OR ("一梯辅助变量".一号梯楼层数 = 3) OR ("一梯辅助变量".一号梯楼层数 = 4);
   "输出变量"."1号梯LEDc" := ("一梯辅助变量".一号梯楼层数 = 1) OR ("一梯辅助变量".一号梯楼层数 = 3) OR ("一梯辅助变量".一号梯楼层数 = 4) OR ("一梯辅助变量".一号梯楼层数 = 5) OR ("一梯辅助变量".一号梯楼层数 = 6);
   "输出变量"."1号梯LEDd" := ("一梯辅助变量".一号梯楼层数 = 2) OR ("一梯辅助变量".一号梯楼层数 = 3) OR ("一梯辅助变量".一号梯楼层数 = 5) OR ("一梯辅助变量".一号梯楼层数 = 6);
   "输出变量"."1号梯LEDe" := ("一梯辅助变量".一号梯楼层数 = 2) OR ("一梯辅助变量".一号梯楼层数 = 6);
   "输出变量"."1号梯LEDf" := ("一梯辅助变量".一号梯楼层数 = 4) OR ("一梯辅助变量".一号梯楼层数 = 5) OR ("一梯辅助变量".一号梯楼层数 = 6);
   "输出变量"."1号梯LEDg" := ("一梯辅助变量".一号梯楼层数 = 2) OR ("一梯辅助变量".一号梯楼层数 = 3) OR ("一梯辅助变量".一号梯楼层数 = 4) OR ("一梯辅助变量".一号梯楼层数 = 5) OR ("一梯辅助变量".一号梯楼层数 = 6);
END_REGION
END_FUNCTION

ORGANIZATION_BLOCK "Main"   // OB1, LAD, ProgramCycle
TITLE = "Main Program Sweep (Cycle)"
{ S7_Optimized_Access := 'TRUE' }
VERSION : 0.1
   VAR_INPUT
      Initial_Call : Bool;   // Initial call of this OB
      Remanence : Bool;   // =True, if remanent data are available
   END_VAR
   VAR_TEMP   // added for the SCL form of the ladder/FBD networks
      _w1 : Bool;
      _w2 : Bool;
      _w3 : Bool;
   END_VAR
BEGIN

REGION Network 1: 未准备就绪则进入初始化,准备就绪后工作
